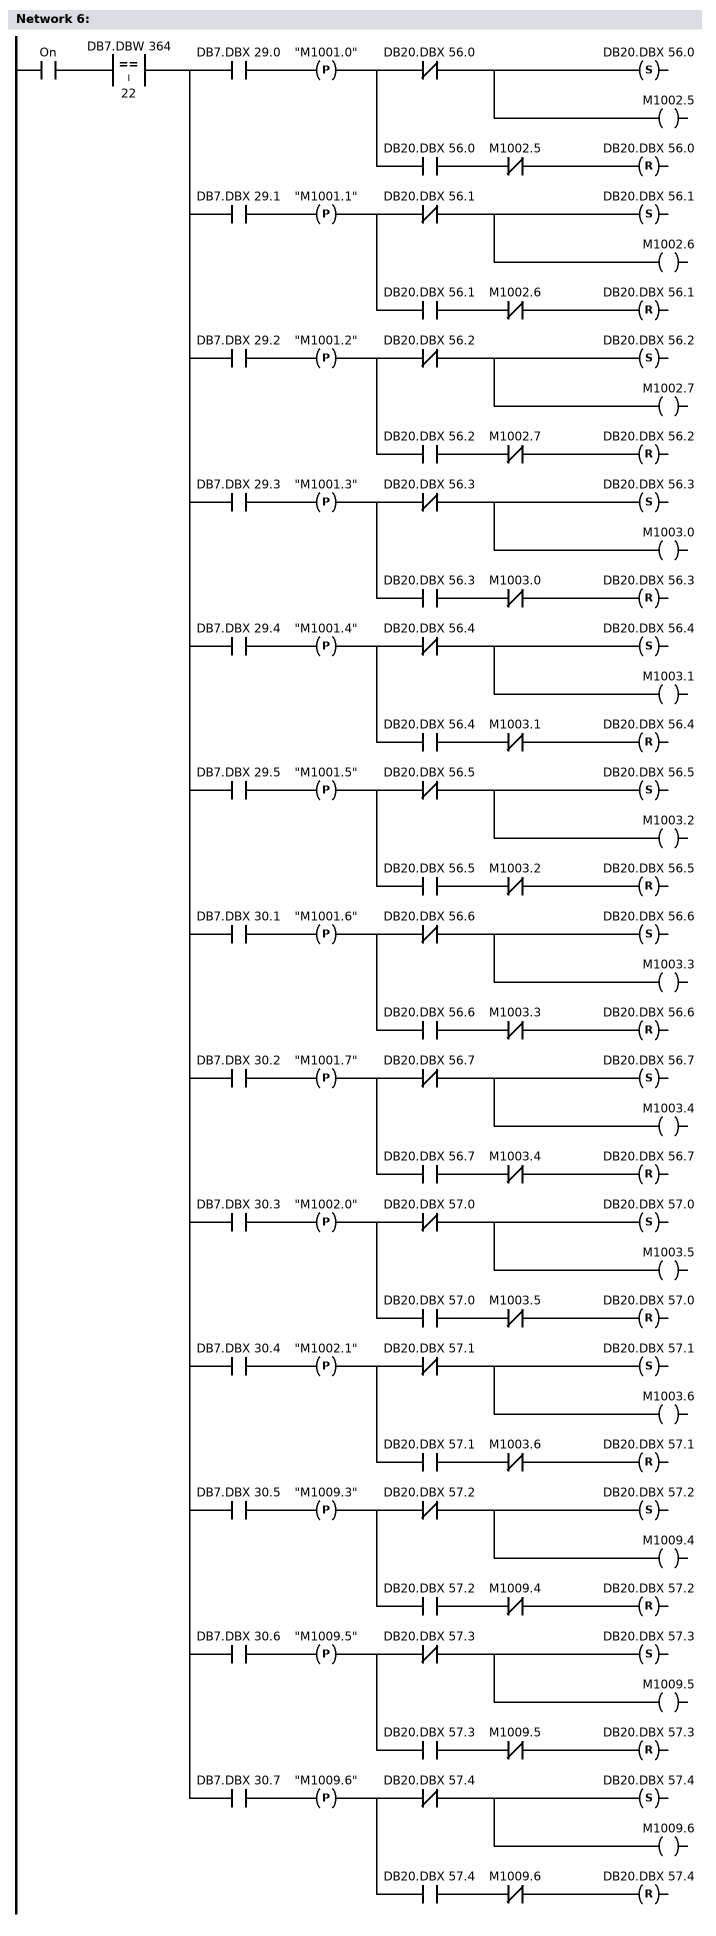
[picture p72: FC53 - REWORK networks 6-6]
NETWORK
TITLE =
      A     "On";
      A(;
      L     DB7.DBW 364;
      L     22;
      ==I;
      );
      =     L 0.0;
      A     L 0.0;
      A     DB7.DBX 29.0;
      FP    "M1001.0";
      =     L 0.1;
      A     L 0.1;
      AN    DB20.DBX 56.0;
      S     DB20.DBX 56.0;
      =     "M1002.5";
      A     L 0.1;
      A     DB20.DBX 56.0;
      AN    "M1002.5";
      R     DB20.DBX 56.0;
      A     L 0.0;
      A     DB7.DBX 29.1;
      FP    "M1001.1";
      =     L 0.1;
      A     L 0.1;
      AN    DB20.DBX 56.1;
      S     DB20.DBX 56.1;
      =     "M1002.6";
      A     L 0.1;
      A     DB20.DBX 56.1;
      AN    "M1002.6";
      R     DB20.DBX 56.1;
      A     L 0.0;
      A     DB7.DBX 29.2;
      FP    "M1001.2";
      =     L 0.1;
      A     L 0.1;
      AN    DB20.DBX 56.2;
      S     DB20.DBX 56.2;
      =     "M1002.7";
      A     L 0.1;
      A     DB20.DBX 56.2;
      AN    "M1002.7";
      R     DB20.DBX 56.2;
      A     L 0.0;
      A     DB7.DBX 29.3;
      FP    "M1001.3";
      =     L 0.1;
      A     L 0.1;
      AN    DB20.DBX 56.3;
      S     DB20.DBX 56.3;
      =     "M1003.0";
      A     L 0.1;
      A     DB20.DBX 56.3;
      AN    "M1003.0";
      R     DB20.DBX 56.3;
      A     L 0.0;
      A     DB7.DBX 29.4;
      FP    "M1001.4";
      =     L 0.1;
      A     L 0.1;
      AN    DB20.DBX 56.4;
      S     DB20.DBX 56.4;
      =     "M1003.1";
      A     L 0.1;
      A     DB20.DBX 56.4;
      AN    "M1003.1";
      R     DB20.DBX 56.4;
      A     L 0.0;
      A     DB7.DBX 29.5;
      FP    "M1001.5";
      =     L 0.1;
      A     L 0.1;
      AN    DB20.DBX 56.5;
      S     DB20.DBX 56.5;
      =     "M1003.2";
      A     L 0.1;
      A     DB20.DBX 56.5;
      AN    "M1003.2";
      R     DB20.DBX 56.5;
      A     L 0.0;
      A     DB7.DBX 30.1;
      FP    "M1001.6";
      =     L 0.1;
      A     L 0.1;
      AN    DB20.DBX 56.6;
      S     DB20.DBX 56.6;
      =     "M1003.3";
      A     L 0.1;
      A     DB20.DBX 56.6;
      AN    "M1003.3";
      R     DB20.DBX 56.6;
      A     L 0.0;
      A     DB7.DBX 30.2;
      FP    "M1001.7";
      =     L 0.1;
      A     L 0.1;
      AN    DB20.DBX 56.7;
      S     DB20.DBX 56.7;
      =     "M1003.4";
      A     L 0.1;
      A     DB20.DBX 56.7;
      AN    "M1003.4";
      R     DB20.DBX 56.7;
      A     L 0.0;
      A     DB7.DBX 30.3;
      FP    "M1002.0";
      =     L 0.1;
      A     L 0.1;
      AN    DB20.DBX 57.0;
      S     DB20.DBX 57.0;
      =     "M1003.5";
      A     L 0.1;
      A     DB20.DBX 57.0;
      AN    "M1003.5";
      R     DB20.DBX 57.0;
      A     L 0.0;
      A     DB7.DBX 30.4;
      FP    "M1002.1";
      =     L 0.1;
      A     L 0.1;
      AN    DB20.DBX 57.1;
      S     DB20.DBX 57.1;
      =     "M1003.6";
      A     L 0.1;
      A     DB20.DBX 57.1;
      AN    "M1003.6";
      R     DB20.DBX 57.1;
      A     L 0.0;
      A     DB7.DBX 30.5;
      FP    "M1009.3";
      =     L 0.1;
      A     L 0.1;
      AN    DB20.DBX 57.2;
      S     DB20.DBX 57.2;
      =     "M1009.4";
      A     L 0.1;
      A     DB20.DBX 57.2;
      AN    "M1009.4";
      R     DB20.DBX 57.2;
      A     L 0.0;
      A     DB7.DBX 30.6;
      FP    "M1009.5";
      =     L 0.1;
      A     L 0.1;
      AN    DB20.DBX 57.3;
      S     DB20.DBX 57.3;
      =     "M1009.5";
      A     L 0.1;
      A     DB20.DBX 57.3;
      AN    "M1009.5";
      R     DB20.DBX 57.3;
      A     L 0.0;
      A     DB7.DBX 30.7;
      FP    "M1009.6";
      =     L 0.1;
      A     L 0.1;
      AN    DB20.DBX 57.4;
      S     DB20.DBX 57.4;
      =     "M1009.6";
      A     L 0.1;
      A     DB20.DBX 57.4;
      AN    "M1009.6";
      R     DB20.DBX 57.4;
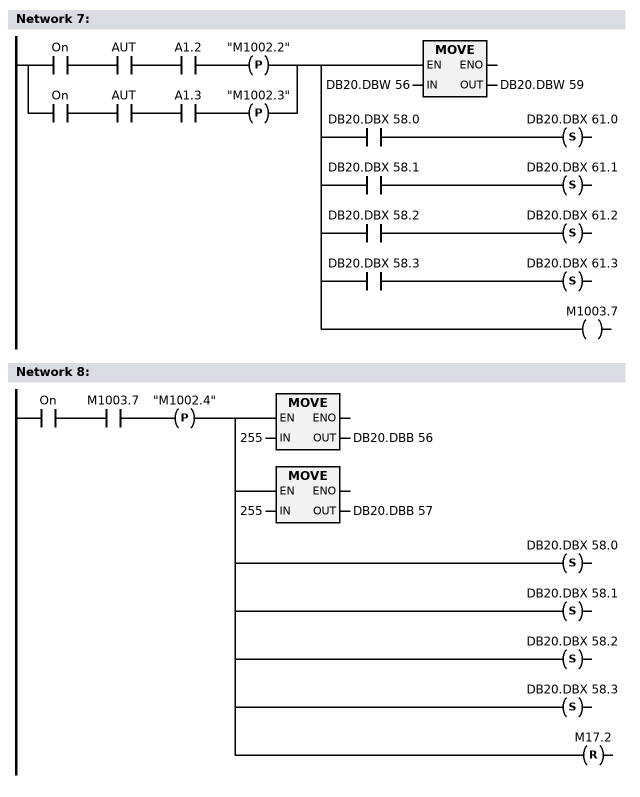
NETWORK
TITLE =
      A     "On";
      A     "AUT";
      A     "A1.2";
      FP    "M1002.2";
      O(;
      A     "On";
      A     "AUT";
      A     "A1.3";
      FP    "M1002.3";
      );
      =     L 0.0;
      A     L 0.0;
      JNB   M009;
      L     DB20.DBW 56;
      T     DB20.DBW 59;
M009: NOP   0;
      A     L 0.0;
      A     DB20.DBX 58.0;
      S     DB20.DBX 61.0;
      A     L 0.0;
      A     DB20.DBX 58.1;
      S     DB20.DBX 61.1;
      A     L 0.0;
      A     DB20.DBX 58.2;
      S     DB20.DBX 61.2;
      A     L 0.0;
      A     DB20.DBX 58.3;
      S     DB20.DBX 61.3;
      A     L 0.0;
      BLD   102;
      =     "M1003.7";
NETWORK
TITLE =
      A     "On";
      A     "M1003.7";
      FP    "M1002.4";
      =     L 0.0;
      A     L 0.0;
      JNB   M010;
      L     255;
      T     DB20.DBB 56;
M010: NOP   0;
      A     L 0.0;
      JNB   M011;
      L     255;
      T     DB20.DBB 57;
M011: NOP   0;
      A     L 0.0;
      BLD   102;
      S     DB20.DBX 58.0;
      A     L 0.0;
      BLD   102;
      S     DB20.DBX 58.1;
      A     L 0.0;
      BLD   102;
      S     DB20.DBX 58.2;
      A     L 0.0;
      BLD   102;
      S     DB20.DBX 58.3;
      A     L 0.0;
      BLD   102;
      R     "M17.2";
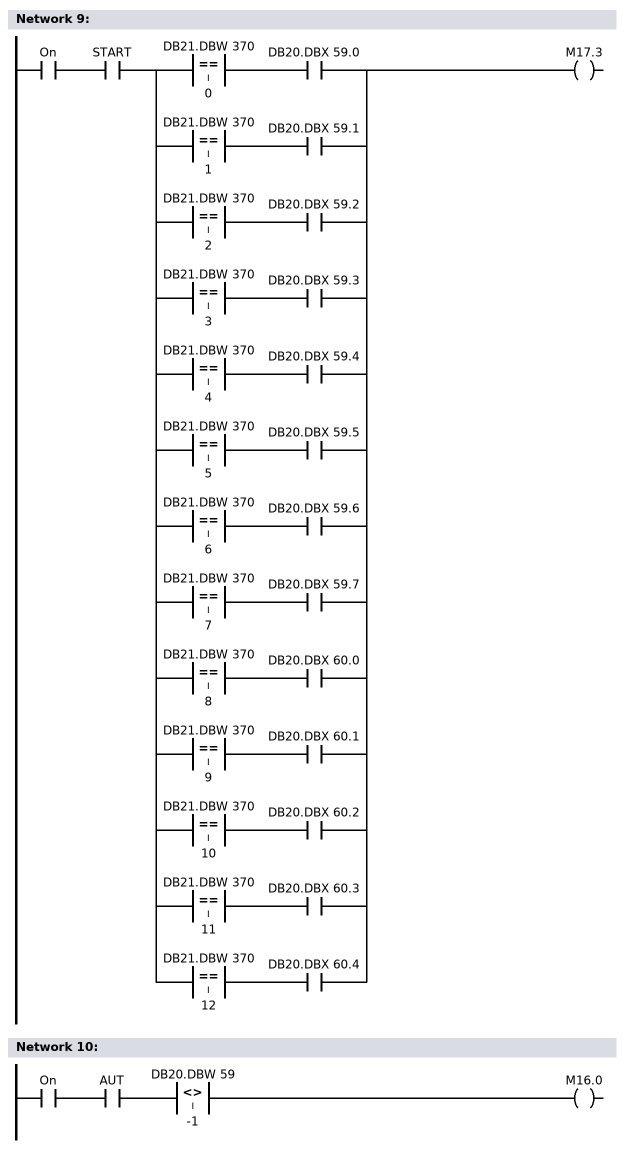
NETWORK
TITLE =
      A     "On";
      A     "START";
      A(;
      A(;
      L     DB21.DBW 370;
      L     0;
      ==I;
      );
      A     DB20.DBX 59.0;
      O;
      A(;
      L     DB21.DBW 370;
      L     1;
      ==I;
      );
      A     DB20.DBX 59.1;
      O;
      A(;
      L     DB21.DBW 370;
      L     2;
      ==I;
      );
      A     DB20.DBX 59.2;
      O;
      A(;
      L     DB21.DBW 370;
      L     3;
      ==I;
      );
      A     DB20.DBX 59.3;
      O;
      A(;
      L     DB21.DBW 370;
      L     4;
      ==I;
      );
      A     DB20.DBX 59.4;
      O;
      A(;
      L     DB21.DBW 370;
      L     5;
      ==I;
      );
      A     DB20.DBX 59.5;
      O;
      A(;
      L     DB21.DBW 370;
      L     6;
      ==I;
      );
      A     DB20.DBX 59.6;
      O;
      A(;
      L     DB21.DBW 370;
      L     7;
      ==I;
      );
      A     DB20.DBX 59.7;
      O;
      A(;
      L     DB21.DBW 370;
      L     8;
      ==I;
      );
      A     DB20.DBX 60.0;
      O;
      A(;
      L     DB21.DBW 370;
      L     9;
      ==I;
      );
      A     DB20.DBX 60.1;
      O;
      A(;
      L     DB21.DBW 370;
      L     10;
      ==I;
      );
      A     DB20.DBX 60.2;
      O;
      A(;
      L     DB21.DBW 370;
      L     11;
      ==I;
      );
      A     DB20.DBX 60.3;
      O;
      A(;
      L     DB21.DBW 370;
      L     12;
      ==I;
      );
      A     DB20.DBX 60.4;
      );
      =     "M17.3";
NETWORK
TITLE =
      A     "On";
      A     "AUT";
      A(;
      L     DB20.DBW 59;
      L     -1;
      <>I;
      );
      =     "M16.0";
END_FUNCTION

FUNCTION FC 54 : VOID
VERSION : 0.1
BEGIN
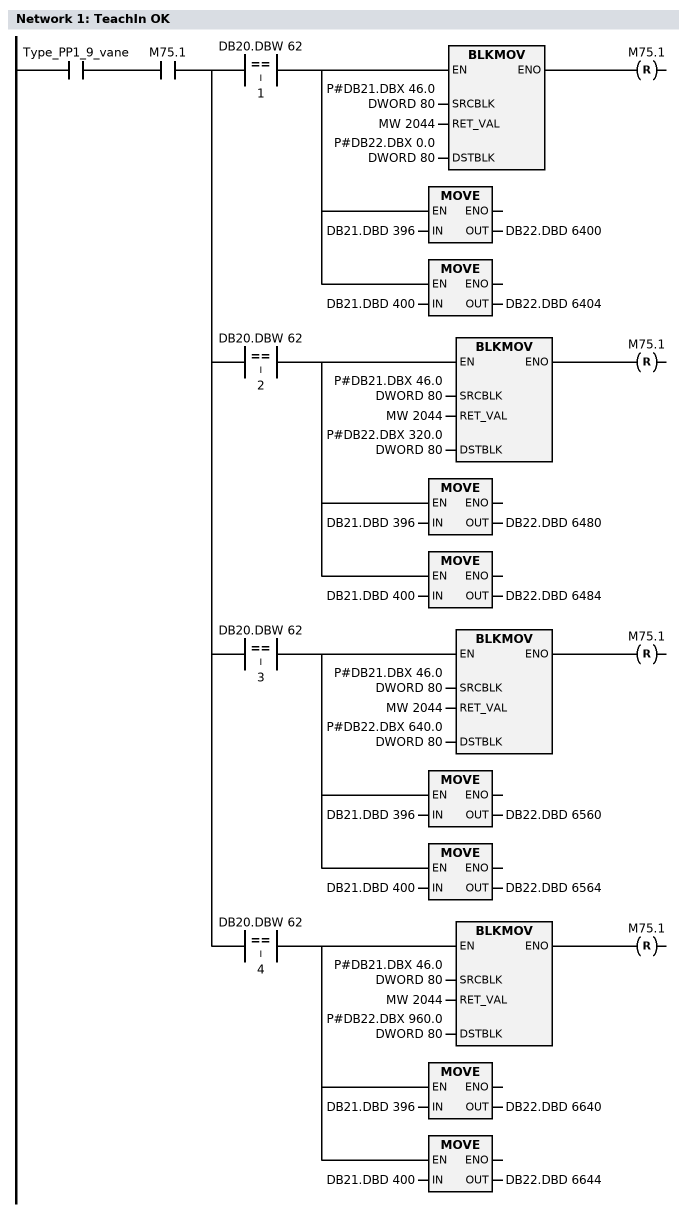
NETWORK
TITLE = TeachIn OK
      A     "Type_PP1_9_vane";
      A     "M75.1";
      =     L 0.0;
      A     L 0.0;
      A(;
      L     DB20.DBW 62;
      L     1;
      ==I;
      );
      =     L 0.1;
      A     L 0.1;
      JNB   _001;
      CALL  "BLKMOV" (
           SRCBLK                   := P#DB21.DBX 46.0 DWORD 80,
           RET_VAL                  := MW 2044,
           DSTBLK                   := P#DB22.DBX 0.0 DWORD 80);
_001: A     BR;
      R     "M75.1";
      A     L 0.1;
      JNB   _002;
      L     DB21.DBD 396;
      T     DB22.DBD 6400;
_002: NOP   0;
      A     L 0.1;
      JNB   _003;
      L     DB21.DBD 400;
      T     DB22.DBD 6404;
_003: NOP   0;
      A     L 0.0;
      A(;
      L     DB20.DBW 62;
      L     2;
      ==I;
      );
      =     L 0.1;
      A     L 0.1;
      JNB   _004;
      CALL  "BLKMOV" (
           SRCBLK                   := P#DB21.DBX 46.0 DWORD 80,
           RET_VAL                  := MW 2044,
           DSTBLK                   := P#DB22.DBX 320.0 DWORD 80);
_004: A     BR;
      R     "M75.1";
      A     L 0.1;
      JNB   _005;
      L     DB21.DBD 396;
      T     DB22.DBD 6480;
_005: NOP   0;
      A     L 0.1;
      JNB   _006;
      L     DB21.DBD 400;
      T     DB22.DBD 6484;
_006: NOP   0;
      A     L 0.0;
      A(;
      L     DB20.DBW 62;
      L     3;
      ==I;
      );
      =     L 0.1;
      A     L 0.1;
      JNB   _007;
      CALL  "BLKMOV" (
           SRCBLK                   := P#DB21.DBX 46.0 DWORD 80,
           RET_VAL                  := MW 2044,
           DSTBLK                   := P#DB22.DBX 640.0 DWORD 80);
_007: A     BR;
      R     "M75.1";
      A     L 0.1;
      JNB   _008;
      L     DB21.DBD 396;
      T     DB22.DBD 6560;
_008: NOP   0;
      A     L 0.1;
      JNB   _009;
      L     DB21.DBD 400;
      T     DB22.DBD 6564;
_009: NOP   0;
      A     L 0.0;
      A(;
      L     DB20.DBW 62;
      L     4;
      ==I;
      );
      =     L 0.1;
      A     L 0.1;
      JNB   _00a;
      CALL  "BLKMOV" (
           SRCBLK                   := P#DB21.DBX 46.0 DWORD 80,
           RET_VAL                  := MW 2044,
           DSTBLK                   := P#DB22.DBX 960.0 DWORD 80);
_00a: A     BR;
      R     "M75.1";
      A     L 0.1;
      JNB   _00b;
      L     DB21.DBD 396;
      T     DB22.DBD 6640;
_00b: NOP   0;
      A     L 0.1;
      JNB   _00c;
      L     DB21.DBD 400;
      T     DB22.DBD 6644;
_00c: NOP   0;
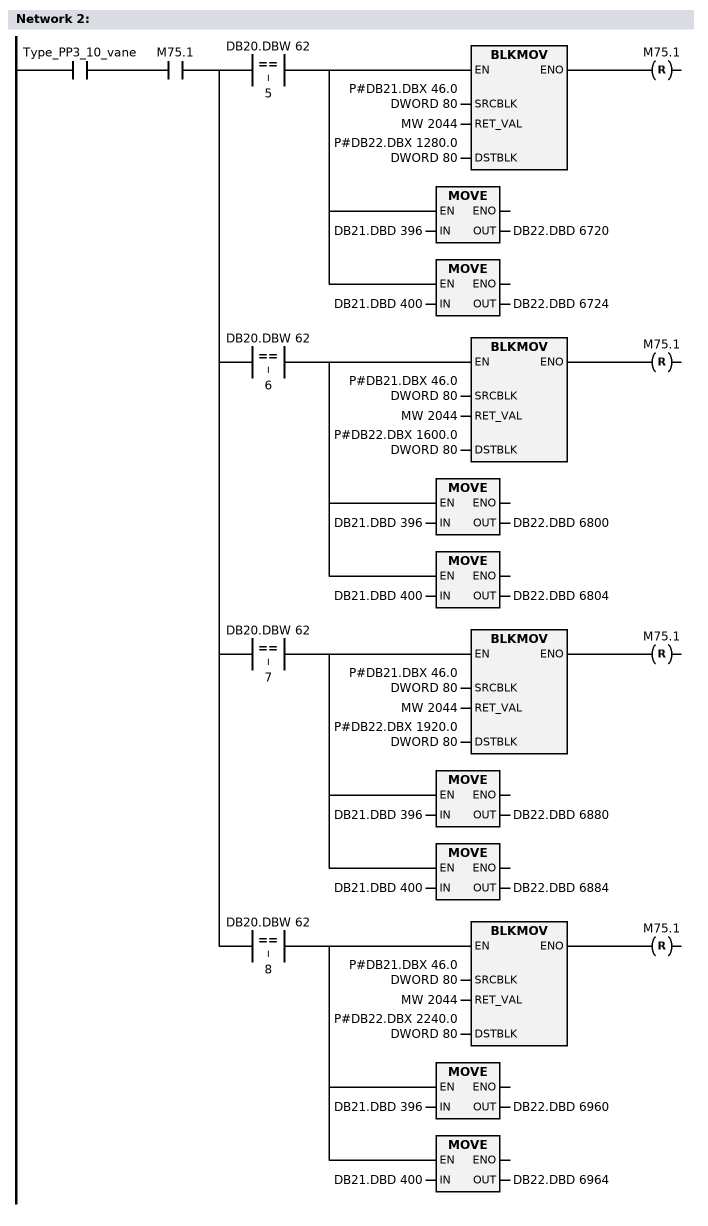
NETWORK
TITLE =
      A     "Type_PP3_10_vane";
      A     "M75.1";
      =     L 0.0;
      A     L 0.0;
      A(;
      L     DB20.DBW 62;
      L     5;
      ==I;
      );
      =     L 0.1;
      A     L 0.1;
      JNB   _00d;
      CALL  "BLKMOV" (
           SRCBLK                   := P#DB21.DBX 46.0 DWORD 80,
           RET_VAL                  := MW 2044,
           DSTBLK                   := P#DB22.DBX 1280.0 DWORD 80);
_00d: A     BR;
      R     "M75.1";
      A     L 0.1;
      JNB   _00e;
      L     DB21.DBD 396;
      T     DB22.DBD 6720;
_00e: NOP   0;
      A     L 0.1;
      JNB   _00f;
      L     DB21.DBD 400;
      T     DB22.DBD 6724;
_00f: NOP   0;
      A     L 0.0;
      A(;
      L     DB20.DBW 62;
      L     6;
      ==I;
      );
      =     L 0.1;
      A     L 0.1;
      JNB   _010;
      CALL  "BLKMOV" (
           SRCBLK                   := P#DB21.DBX 46.0 DWORD 80,
           RET_VAL                  := MW 2044,
           DSTBLK                   := P#DB22.DBX 1600.0 DWORD 80);
_010: A     BR;
      R     "M75.1";
      A     L 0.1;
      JNB   _011;
      L     DB21.DBD 396;
      T     DB22.DBD 6800;
_011: NOP   0;
      A     L 0.1;
      JNB   _012;
      L     DB21.DBD 400;
      T     DB22.DBD 6804;
_012: NOP   0;
      A     L 0.0;
      A(;
      L     DB20.DBW 62;
      L     7;
      ==I;
      );
      =     L 0.1;
      A     L 0.1;
      JNB   _013;
      CALL  "BLKMOV" (
           SRCBLK                   := P#DB21.DBX 46.0 DWORD 80,
           RET_VAL                  := MW 2044,
           DSTBLK                   := P#DB22.DBX 1920.0 DWORD 80);
_013: A     BR;
      R     "M75.1";
      A     L 0.1;
      JNB   _014;
      L     DB21.DBD 396;
      T     DB22.DBD 6880;
_014: NOP   0;
      A     L 0.1;
      JNB   _015;
      L     DB21.DBD 400;
      T     DB22.DBD 6884;
_015: NOP   0;
      A     L 0.0;
      A(;
      L     DB20.DBW 62;
      L     8;
      ==I;
      );
      =     L 0.1;
      A     L 0.1;
      JNB   _016;
      CALL  "BLKMOV" (
           SRCBLK                   := P#DB21.DBX 46.0 DWORD 80,
           RET_VAL                  := MW 2044,
           DSTBLK                   := P#DB22.DBX 2240.0 DWORD 80);
_016: A     BR;
      R     "M75.1";
      A     L 0.1;
      JNB   _017;
      L     DB21.DBD 396;
      T     DB22.DBD 6960;
_017: NOP   0;
      A     L 0.1;
      JNB   _018;
      L     DB21.DBD 400;
      T     DB22.DBD 6964;
_018: NOP   0;
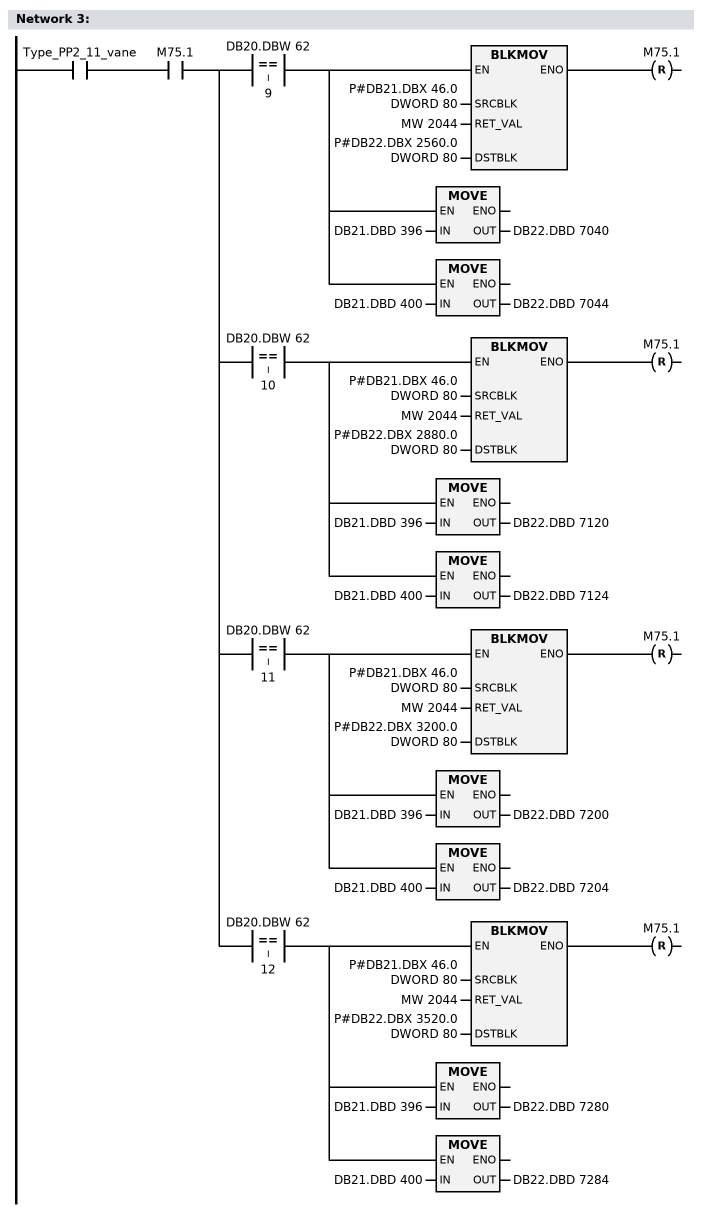
NETWORK
TITLE =
      A     "Type_PP2_11_vane";
      A     "M75.1";
      =     L 0.0;
      A     L 0.0;
      A(;
      L     DB20.DBW 62;
      L     9;
      ==I;
      );
      =     L 0.1;
      A     L 0.1;
      JNB   _019;
      CALL  "BLKMOV" (
           SRCBLK                   := P#DB21.DBX 46.0 DWORD 80,
           RET_VAL                  := MW 2044,
           DSTBLK                   := P#DB22.DBX 2560.0 DWORD 80);
_019: A     BR;
      R     "M75.1";
      A     L 0.1;
      JNB   _01a;
      L     DB21.DBD 396;
      T     DB22.DBD 7040;
_01a: NOP   0;
      A     L 0.1;
      JNB   _01b;
      L     DB21.DBD 400;
      T     DB22.DBD 7044;
_01b: NOP   0;
      A     L 0.0;
      A(;
      L     DB20.DBW 62;
      L     10;
      ==I;
      );
      =     L 0.1;
      A     L 0.1;
      JNB   _01c;
      CALL  "BLKMOV" (
           SRCBLK                   := P#DB21.DBX 46.0 DWORD 80,
           RET_VAL                  := MW 2044,
           DSTBLK                   := P#DB22.DBX 2880.0 DWORD 80);
_01c: A     BR;
      R     "M75.1";
      A     L 0.1;
      JNB   _01d;
      L     DB21.DBD 396;
      T     DB22.DBD 7120;
_01d: NOP   0;
      A     L 0.1;
      JNB   _01e;
      L     DB21.DBD 400;
      T     DB22.DBD 7124;
_01e: NOP   0;
      A     L 0.0;
      A(;
      L     DB20.DBW 62;
      L     11;
      ==I;
      );
      =     L 0.1;
      A     L 0.1;
      JNB   _01f;
      CALL  "BLKMOV" (
           SRCBLK                   := P#DB21.DBX 46.0 DWORD 80,
           RET_VAL                  := MW 2044,
           DSTBLK                   := P#DB22.DBX 3200.0 DWORD 80);
_01f: A     BR;
      R     "M75.1";
      A     L 0.1;
      JNB   _020;
      L     DB21.DBD 396;
      T     DB22.DBD 7200;
_020: NOP   0;
      A     L 0.1;
      JNB   _021;
      L     DB21.DBD 400;
      T     DB22.DBD 7204;
_021: NOP   0;
      A     L 0.0;
      A(;
      L     DB20.DBW 62;
      L     12;
      ==I;
      );
      =     L 0.1;
      A     L 0.1;
      JNB   _022;
      CALL  "BLKMOV" (
           SRCBLK                   := P#DB21.DBX 46.0 DWORD 80,
           RET_VAL                  := MW 2044,
           DSTBLK                   := P#DB22.DBX 3520.0 DWORD 80);
_022: A     BR;
      R     "M75.1";
      A     L 0.1;
      JNB   _023;
      L     DB21.DBD 396;
      T     DB22.DBD 7280;
_023: NOP   0;
      A     L 0.1;
      JNB   _024;
      L     DB21.DBD 400;
      T     DB22.DBD 7284;
_024: NOP   0;
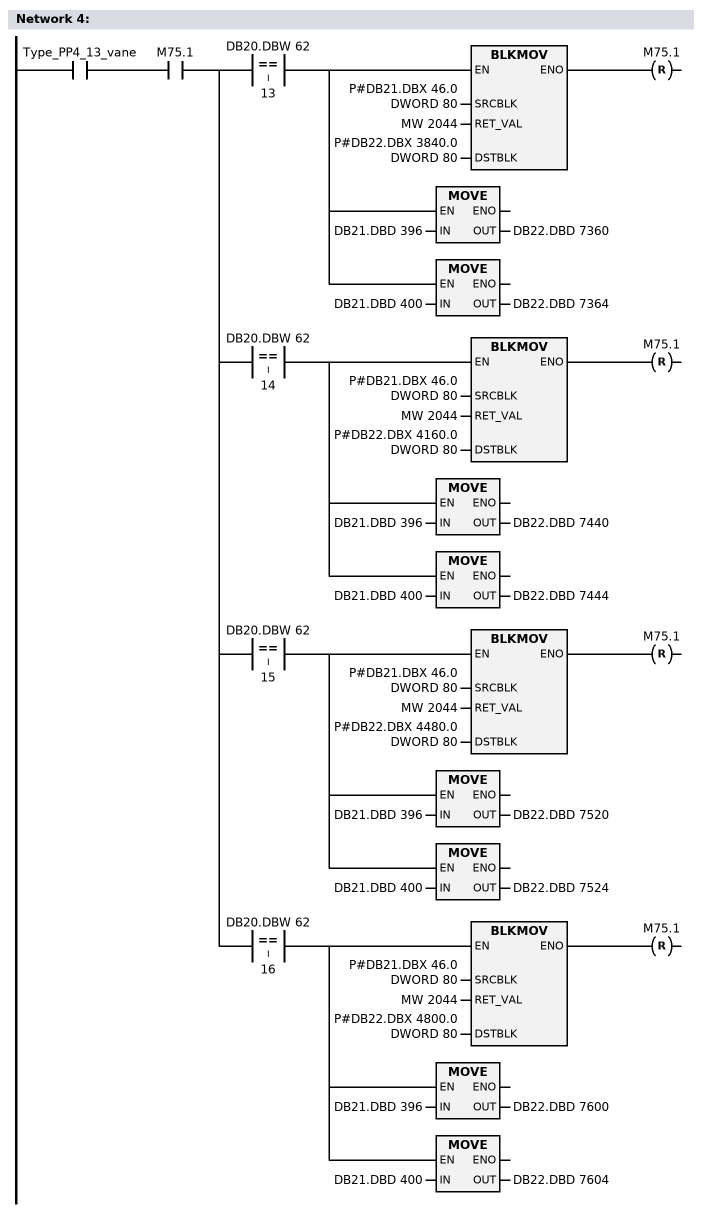
NETWORK
TITLE =
      A     "Type_PP4_13_vane";
      A     "M75.1";
      =     L 0.0;
      A     L 0.0;
      A(;
      L     DB20.DBW 62;
      L     13;
      ==I;
      );
      =     L 0.1;
      A     L 0.1;
      JNB   _025;
      CALL  "BLKMOV" (
           SRCBLK                   := P#DB21.DBX 46.0 DWORD 80,
           RET_VAL                  := MW 2044,
           DSTBLK                   := P#DB22.DBX 3840.0 DWORD 80);
_025: A     BR;
      R     "M75.1";
      A     L 0.1;
      JNB   _026;
      L     DB21.DBD 396;
      T     DB22.DBD 7360;
_026: NOP   0;
      A     L 0.1;
      JNB   _027;
      L     DB21.DBD 400;
      T     DB22.DBD 7364;
_027: NOP   0;
      A     L 0.0;
      A(;
      L     DB20.DBW 62;
      L     14;
      ==I;
      );
      =     L 0.1;
      A     L 0.1;
      JNB   _028;
      CALL  "BLKMOV" (
           SRCBLK                   := P#DB21.DBX 46.0 DWORD 80,
           RET_VAL                  := MW 2044,
           DSTBLK                   := P#DB22.DBX 4160.0 DWORD 80);
_028: A     BR;
      R     "M75.1";
      A     L 0.1;
      JNB   _029;
      L     DB21.DBD 396;
      T     DB22.DBD 7440;
_029: NOP   0;
      A     L 0.1;
      JNB   _02a;
      L     DB21.DBD 400;
      T     DB22.DBD 7444;
_02a: NOP   0;
      A     L 0.0;
      A(;
      L     DB20.DBW 62;
      L     15;
      ==I;
      );
      =     L 0.1;
      A     L 0.1;
      JNB   _02b;
      CALL  "BLKMOV" (
           SRCBLK                   := P#DB21.DBX 46.0 DWORD 80,
           RET_VAL                  := MW 2044,
           DSTBLK                   := P#DB22.DBX 4480.0 DWORD 80);
_02b: A     BR;
      R     "M75.1";
      A     L 0.1;
      JNB   _02c;
      L     DB21.DBD 396;
      T     DB22.DBD 7520;
_02c: NOP   0;
      A     L 0.1;
      JNB   _02d;
      L     DB21.DBD 400;
      T     DB22.DBD 7524;
_02d: NOP   0;
      A     L 0.0;
      A(;
      L     DB20.DBW 62;
      L     16;
      ==I;
      );
      =     L 0.1;
      A     L 0.1;
      JNB   _02e;
      CALL  "BLKMOV" (
           SRCBLK                   := P#DB21.DBX 46.0 DWORD 80,
           RET_VAL                  := MW 2044,
           DSTBLK                   := P#DB22.DBX 4800.0 DWORD 80);
_02e: A     BR;
      R     "M75.1";
      A     L 0.1;
      JNB   _02f;
      L     DB21.DBD 396;
      T     DB22.DBD 7600;
_02f: NOP   0;
      A     L 0.1;
      JNB   _030;
      L     DB21.DBD 400;
      T     DB22.DBD 7604;
_030: NOP   0;
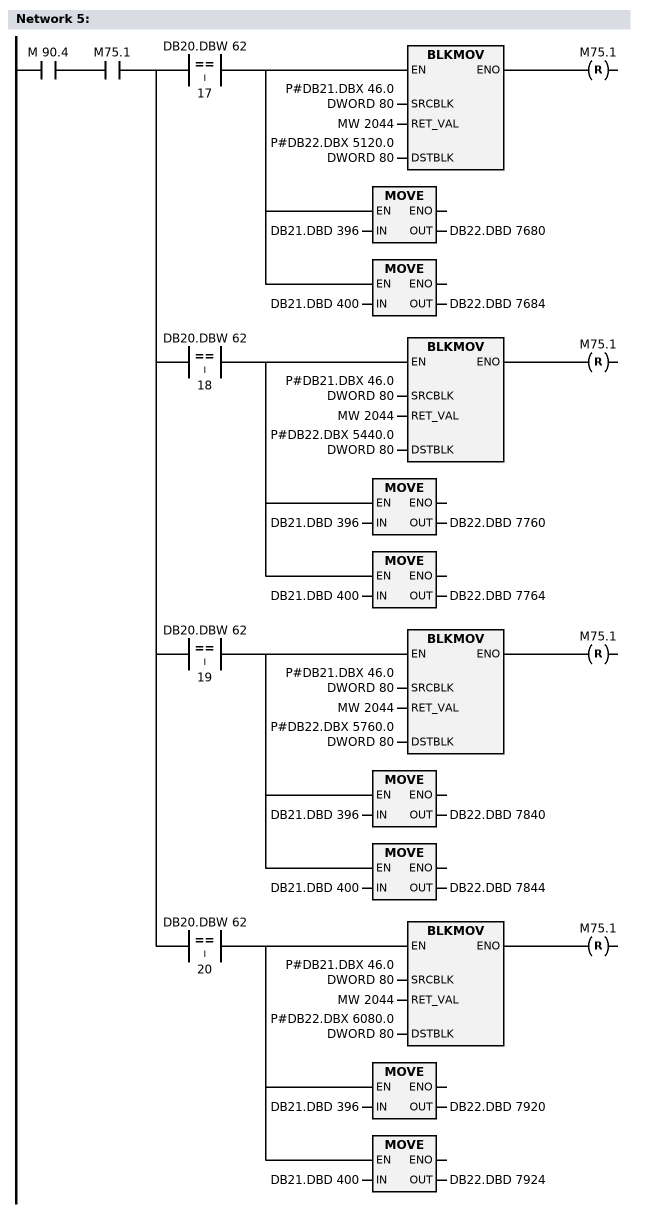
NETWORK
TITLE =
      A     M 90.4;
      A     "M75.1";
      =     L 0.0;
      A     L 0.0;
      A(;
      L     DB20.DBW 62;
      L     17;
      ==I;
      );
      =     L 0.1;
      A     L 0.1;
      JNB   _031;
      CALL  "BLKMOV" (
           SRCBLK                   := P#DB21.DBX 46.0 DWORD 80,
           RET_VAL                  := MW 2044,
           DSTBLK                   := P#DB22.DBX 5120.0 DWORD 80);
_031: A     BR;
      R     "M75.1";
      A     L 0.1;
      JNB   _032;
      L     DB21.DBD 396;
      T     DB22.DBD 7680;
_032: NOP   0;
      A     L 0.1;
      JNB   _033;
      L     DB21.DBD 400;
      T     DB22.DBD 7684;
_033: NOP   0;
      A     L 0.0;
      A(;
      L     DB20.DBW 62;
      L     18;
      ==I;
      );
      =     L 0.1;
      A     L 0.1;
      JNB   _034;
      CALL  "BLKMOV" (
           SRCBLK                   := P#DB21.DBX 46.0 DWORD 80,
           RET_VAL                  := MW 2044,
           DSTBLK                   := P#DB22.DBX 5440.0 DWORD 80);
_034: A     BR;
      R     "M75.1";
      A     L 0.1;
      JNB   _035;
      L     DB21.DBD 396;
      T     DB22.DBD 7760;
_035: NOP   0;
      A     L 0.1;
      JNB   _036;
      L     DB21.DBD 400;
      T     DB22.DBD 7764;
_036: NOP   0;
      A     L 0.0;
      A(;
      L     DB20.DBW 62;
      L     19;
      ==I;
      );
      =     L 0.1;
      A     L 0.1;
      JNB   _037;
      CALL  "BLKMOV" (
           SRCBLK                   := P#DB21.DBX 46.0 DWORD 80,
           RET_VAL                  := MW 2044,
           DSTBLK                   := P#DB22.DBX 5760.0 DWORD 80);
_037: A     BR;
      R     "M75.1";
      A     L 0.1;
      JNB   _038;
      L     DB21.DBD 396;
      T     DB22.DBD 7840;
_038: NOP   0;
      A     L 0.1;
      JNB   _039;
      L     DB21.DBD 400;
      T     DB22.DBD 7844;
_039: NOP   0;
      A     L 0.0;
      A(;
      L     DB20.DBW 62;
      L     20;
      ==I;
      );
      =     L 0.1;
      A     L 0.1;
      JNB   _03a;
      CALL  "BLKMOV" (
           SRCBLK                   := P#DB21.DBX 46.0 DWORD 80,
           RET_VAL                  := MW 2044,
           DSTBLK                   := P#DB22.DBX 6080.0 DWORD 80);
_03a: A     BR;
      R     "M75.1";
      A     L 0.1;
      JNB   _03b;
      L     DB21.DBD 396;
      T     DB22.DBD 7920;
_03b: NOP   0;
      A     L 0.1;
      JNB   _03c;
      L     DB21.DBD 400;
      T     DB22.DBD 7924;
_03c: NOP   0;
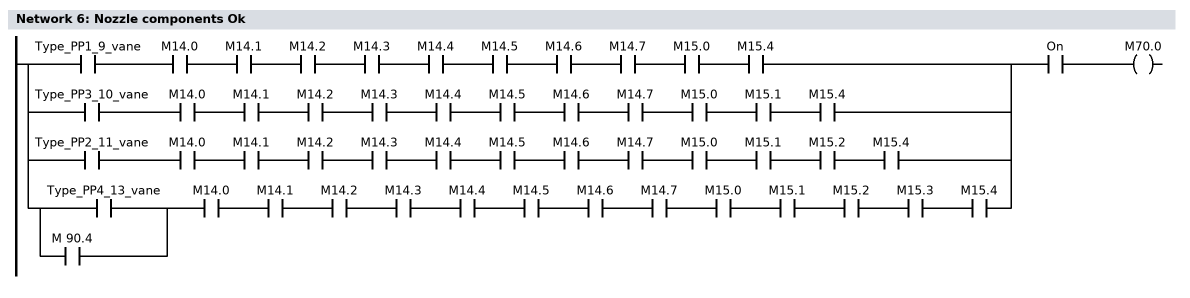
NETWORK
TITLE = Nozzle components Ok
      A(;
      A     "Type_PP1_9_vane";
      A     "M14.0";
      A     "M14.1";
      A     "M14.2";
      A     "M14.3";
      A     "M14.4";
      A     "M14.5";
      A     "M14.6";
      A     "M14.7";
      A     "M15.0";
      A     "M15.4";
      O;
      A     "Type_PP3_10_vane";
      A     "M14.0";
      A     "M14.1";
      A     "M14.2";
      A     "M14.3";
      A     "M14.4";
      A     "M14.5";
      A     "M14.6";
      A     "M14.7";
      A     "M15.0";
      A     "M15.1";
      A     "M15.4";
      O;
      A     "Type_PP2_11_vane";
      A     "M14.0";
      A     "M14.1";
      A     "M14.2";
      A     "M14.3";
      A     "M14.4";
      A     "M14.5";
      A     "M14.6";
      A     "M14.7";
      A     "M15.0";
      A     "M15.1";
      A     "M15.2";
      A     "M15.4";
      O;
      A(;
      O     "Type_PP4_13_vane";
      O     M 90.4;
      );
      A     "M14.0";
      A     "M14.1";
      A     "M14.2";
      A     "M14.3";
      A     "M14.4";
      A     "M14.5";
      A     "M14.6";
      A     "M14.7";
      A     "M15.0";
      A     "M15.1";
      A     "M15.2";
      A     "M15.3";
      A     "M15.4";
      );
      A     "On";
      =     "M70.0";
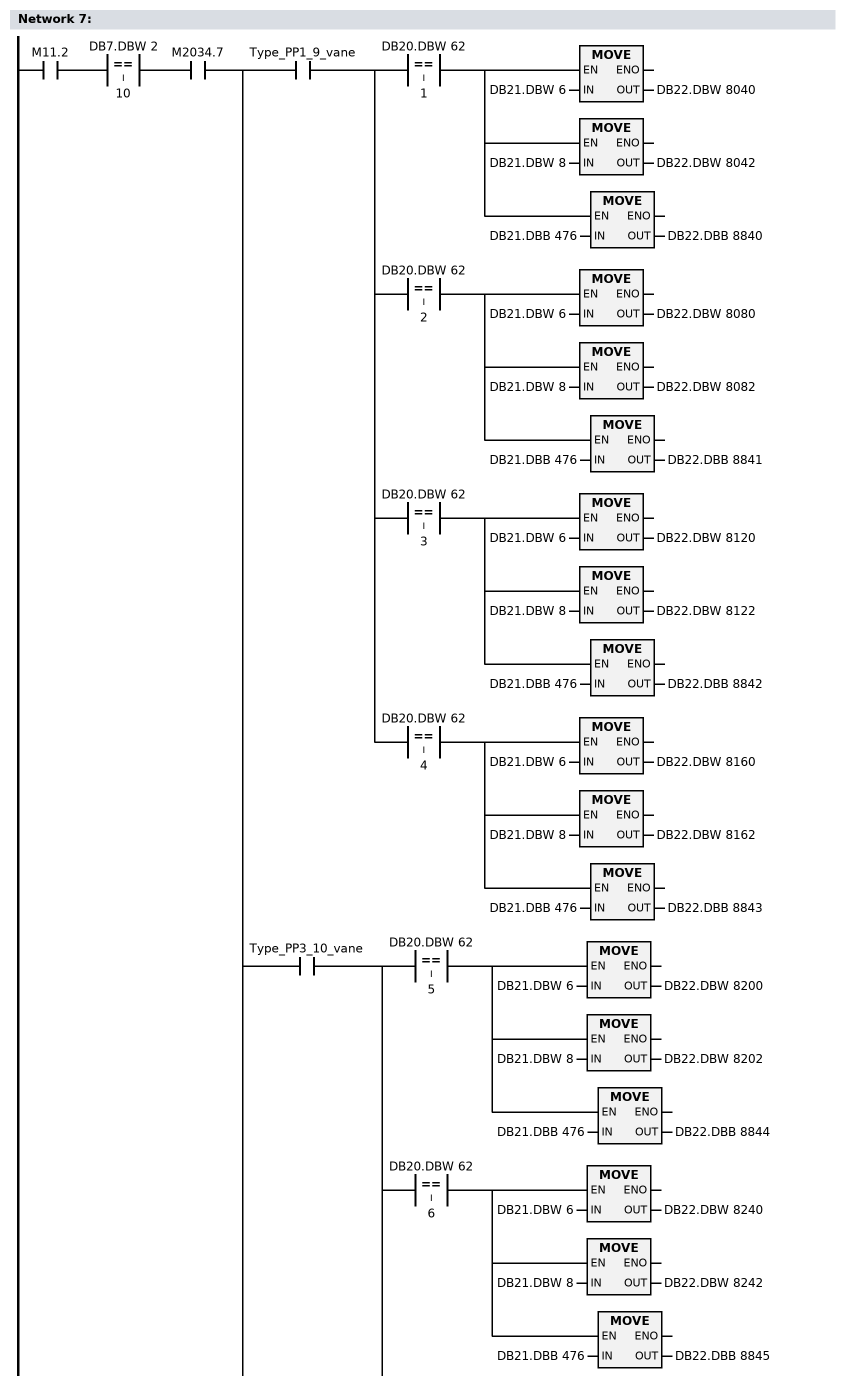
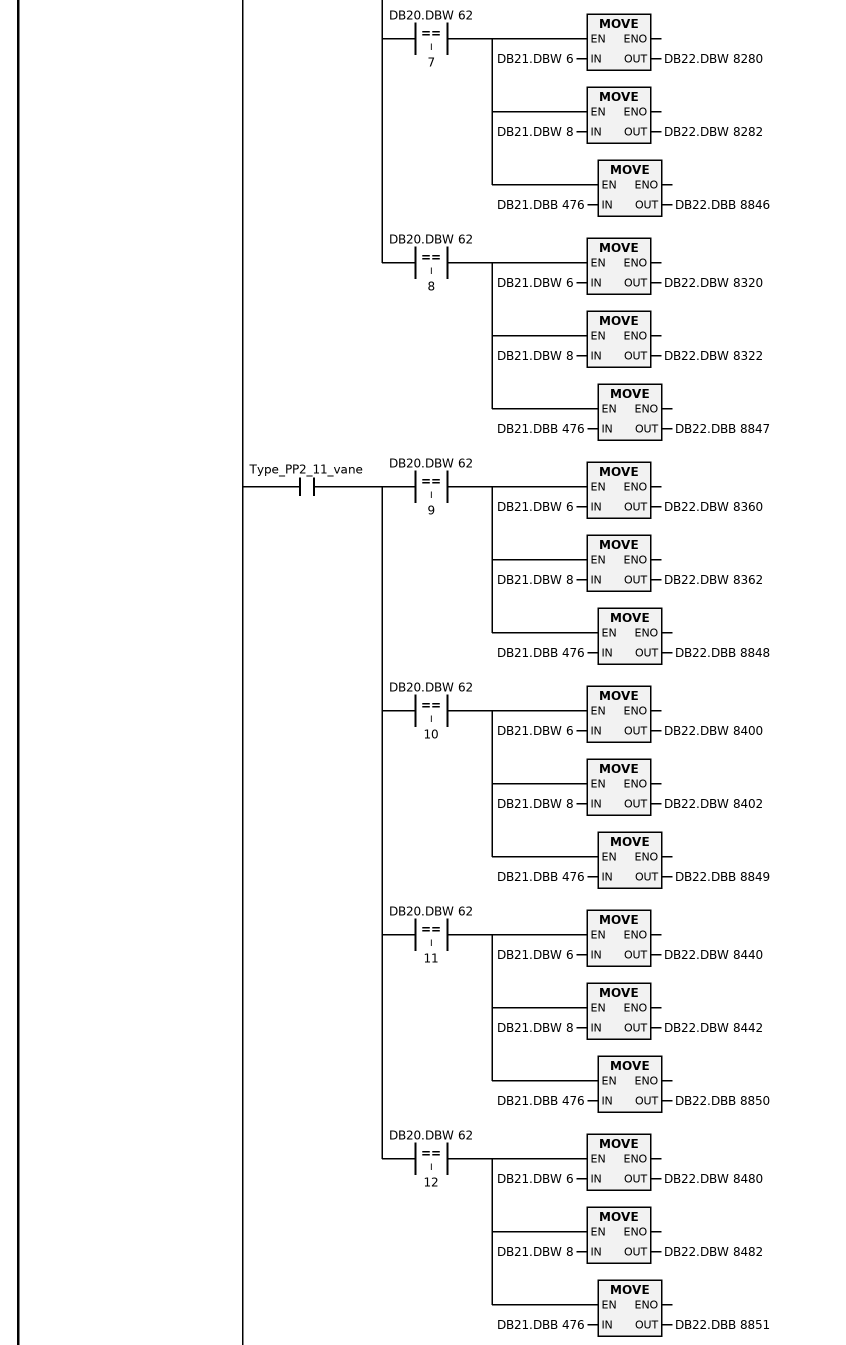
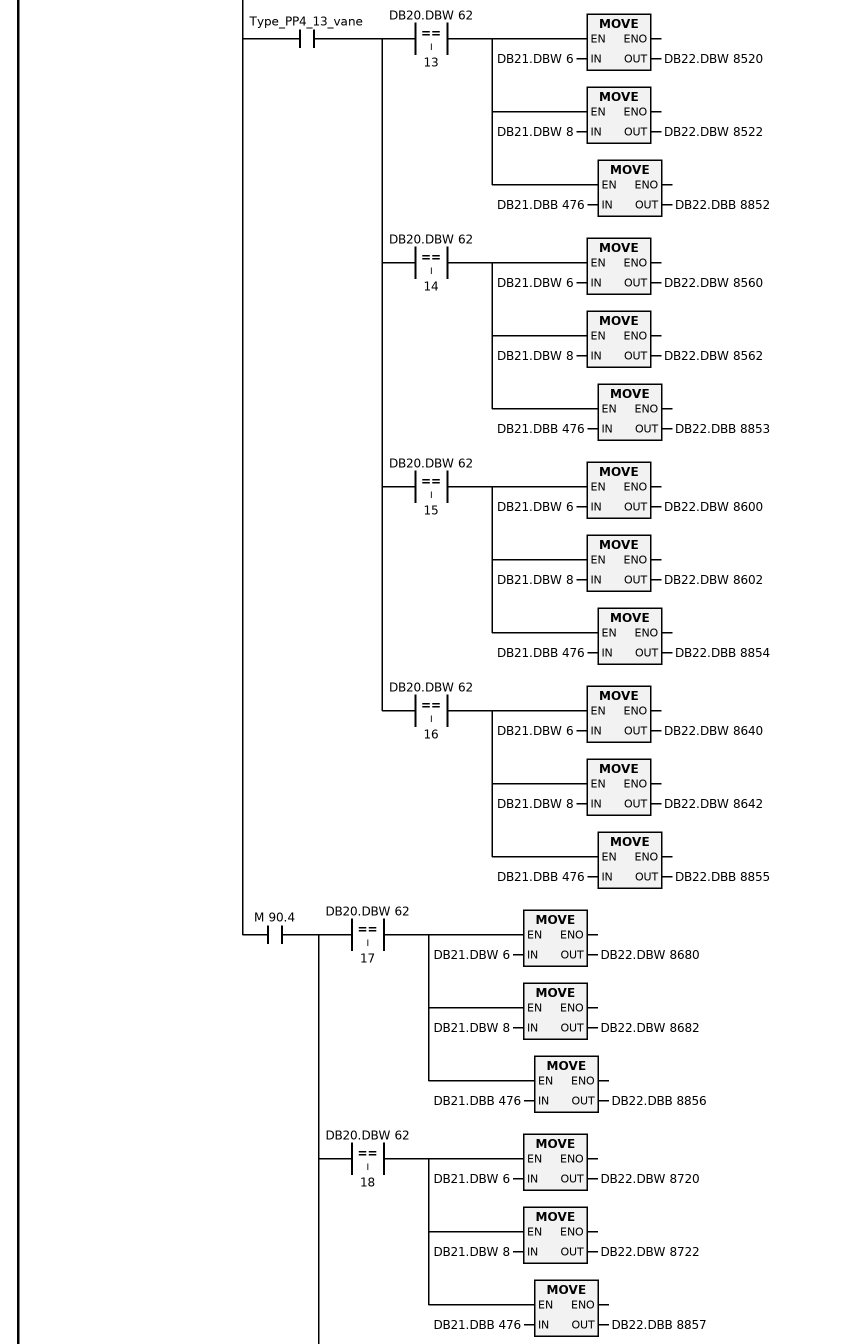
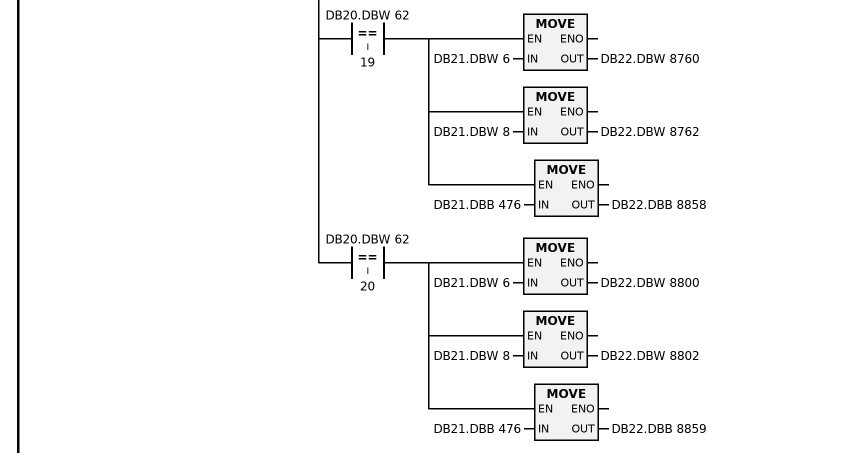
NETWORK
TITLE =
      A     "M11.2";
      A(;
      L     DB7.DBW 2;
      L     10;
      ==I;
      );
      A     "M2034.7";
      =     L 0.0;
      A     L 0.0;
      A     "Type_PP1_9_vane";
      =     L 0.1;
      A     L 0.1;
      A(;
      L     DB20.DBW 62;
      L     1;
      ==I;
      );
      =     L 0.2;
      A     L 0.2;
      JNB   _03d;
      L     DB21.DBW 6;
      T     DB22.DBW 8040;
_03d: NOP   0;
      A     L 0.2;
      JNB   _03e;
      L     DB21.DBW 8;
      T     DB22.DBW 8042;
_03e: NOP   0;
      A     L 0.2;
      JNB   _03f;
      L     DB21.DBB 476;
      T     DB22.DBB 8840;
_03f: NOP   0;
      A     L 0.1;
      A(;
      L     DB20.DBW 62;
      L     2;
      ==I;
      );
      =     L 0.2;
      A     L 0.2;
      JNB   _040;
      L     DB21.DBW 6;
      T     DB22.DBW 8080;
_040: NOP   0;
      A     L 0.2;
      JNB   _041;
      L     DB21.DBW 8;
      T     DB22.DBW 8082;
_041: NOP   0;
      A     L 0.2;
      JNB   _042;
      L     DB21.DBB 476;
      T     DB22.DBB 8841;
_042: NOP   0;
      A     L 0.1;
      A(;
      L     DB20.DBW 62;
      L     3;
      ==I;
      );
      =     L 0.2;
      A     L 0.2;
      JNB   _043;
      L     DB21.DBW 6;
      T     DB22.DBW 8120;
_043: NOP   0;
      A     L 0.2;
      JNB   _044;
      L     DB21.DBW 8;
      T     DB22.DBW 8122;
_044: NOP   0;
      A     L 0.2;
      JNB   _045;
      L     DB21.DBB 476;
      T     DB22.DBB 8842;
_045: NOP   0;
      A     L 0.1;
      A(;
      L     DB20.DBW 62;
      L     4;
      ==I;
      );
      =     L 0.2;
      A     L 0.2;
      JNB   _046;
      L     DB21.DBW 6;
      T     DB22.DBW 8160;
_046: NOP   0;
      A     L 0.2;
      JNB   _047;
      L     DB21.DBW 8;
      T     DB22.DBW 8162;
_047: NOP   0;
      A     L 0.2;
      JNB   _048;
      L     DB21.DBB 476;
      T     DB22.DBB 8843;
_048: NOP   0;
      A     L 0.0;
      A     "Type_PP3_10_vane";
      =     L 0.1;
      A     L 0.1;
      A(;
      L     DB20.DBW 62;
      L     5;
      ==I;
      );
      =     L 0.2;
      A     L 0.2;
      JNB   _049;
      L     DB21.DBW 6;
      T     DB22.DBW 8200;
_049: NOP   0;
      A     L 0.2;
      JNB   _04a;
      L     DB21.DBW 8;
      T     DB22.DBW 8202;
_04a: NOP   0;
      A     L 0.2;
      JNB   _04b;
      L     DB21.DBB 476;
      T     DB22.DBB 8844;
_04b: NOP   0;
      A     L 0.1;
      A(;
      L     DB20.DBW 62;
      L     6;
      ==I;
      );
      =     L 0.2;
      A     L 0.2;
      JNB   _04c;
      L     DB21.DBW 6;
      T     DB22.DBW 8240;
_04c: NOP   0;
      A     L 0.2;
      JNB   _04d;
      L     DB21.DBW 8;
      T     DB22.DBW 8242;
_04d: NOP   0;
      A     L 0.2;
      JNB   _04e;
      L     DB21.DBB 476;
      T     DB22.DBB 8845;
_04e: NOP   0;
      A     L 0.1;
      A(;
      L     DB20.DBW 62;
      L     7;
      ==I;
      );
      =     L 0.2;
      A     L 0.2;
      JNB   _04f;
      L     DB21.DBW 6;
      T     DB22.DBW 8280;
_04f: NOP   0;
      A     L 0.2;
      JNB   _050;
      L     DB21.DBW 8;
      T     DB22.DBW 8282;
_050: NOP   0;
      A     L 0.2;
      JNB   _051;
      L     DB21.DBB 476;
      T     DB22.DBB 8846;
_051: NOP   0;
      A     L 0.1;
      A(;
      L     DB20.DBW 62;
      L     8;
      ==I;
      );
      =     L 0.2;
      A     L 0.2;
      JNB   _052;
      L     DB21.DBW 6;
      T     DB22.DBW 8320;
_052: NOP   0;
      A     L 0.2;
      JNB   _053;
      L     DB21.DBW 8;
      T     DB22.DBW 8322;
_053: NOP   0;
      A     L 0.2;
      JNB   _054;
      L     DB21.DBB 476;
      T     DB22.DBB 8847;
_054: NOP   0;
      A     L 0.0;
      A     "Type_PP2_11_vane";
      =     L 0.1;
      A     L 0.1;
      A(;
      L     DB20.DBW 62;
      L     9;
      ==I;
      );
      =     L 0.2;
      A     L 0.2;
      JNB   _055;
      L     DB21.DBW 6;
      T     DB22.DBW 8360;
_055: NOP   0;
      A     L 0.2;
      JNB   _056;
      L     DB21.DBW 8;
      T     DB22.DBW 8362;
_056: NOP   0;
      A     L 0.2;
      JNB   _057;
      L     DB21.DBB 476;
      T     DB22.DBB 8848;
_057: NOP   0;
      A     L 0.1;
      A(;
      L     DB20.DBW 62;
      L     10;
      ==I;
      );
      =     L 0.2;
      A     L 0.2;
      JNB   _058;
      L     DB21.DBW 6;
      T     DB22.DBW 8400;
_058: NOP   0;
      A     L 0.2;
      JNB   _059;
      L     DB21.DBW 8;
      T     DB22.DBW 8402;
_059: NOP   0;
      A     L 0.2;
      JNB   _05a;
      L     DB21.DBB 476;
      T     DB22.DBB 8849;
_05a: NOP   0;
      A     L 0.1;
      A(;
      L     DB20.DBW 62;
      L     11;
      ==I;
      );
      =     L 0.2;
      A     L 0.2;
      JNB   _05b;
      L     DB21.DBW 6;
      T     DB22.DBW 8440;
_05b: NOP   0;
      A     L 0.2;
      JNB   _05c;
      L     DB21.DBW 8;
      T     DB22.DBW 8442;
_05c: NOP   0;
      A     L 0.2;
      JNB   _05d;
      L     DB21.DBB 476;
      T     DB22.DBB 8850;
_05d: NOP   0;
      A     L 0.1;
      A(;
      L     DB20.DBW 62;
      L     12;
      ==I;
      );
      =     L 0.2;
      A     L 0.2;
      JNB   _05e;
      L     DB21.DBW 6;
      T     DB22.DBW 8480;
_05e: NOP   0;
      A     L 0.2;
      JNB   _05f;
      L     DB21.DBW 8;
      T     DB22.DBW 8482;
_05f: NOP   0;
      A     L 0.2;
      JNB   _060;
      L     DB21.DBB 476;
      T     DB22.DBB 8851;
_060: NOP   0;
      A     L 0.0;
      A     "Type_PP4_13_vane";
      =     L 0.1;
      A     L 0.1;
      A(;
      L     DB20.DBW 62;
      L     13;
      ==I;
      );
      =     L 0.2;
      A     L 0.2;
      JNB   _061;
      L     DB21.DBW 6;
      T     DB22.DBW 8520;
_061: NOP   0;
      A     L 0.2;
      JNB   _062;
      L     DB21.DBW 8;
      T     DB22.DBW 8522;
_062: NOP   0;
      A     L 0.2;
      JNB   _063;
      L     DB21.DBB 476;
      T     DB22.DBB 8852;
_063: NOP   0;
      A     L 0.1;
      A(;
      L     DB20.DBW 62;
      L     14;
      ==I;
      );
      =     L 0.2;
      A     L 0.2;
      JNB   _064;
      L     DB21.DBW 6;
      T     DB22.DBW 8560;
_064: NOP   0;
      A     L 0.2;
      JNB   _065;
      L     DB21.DBW 8;
      T     DB22.DBW 8562;
_065: NOP   0;
      A     L 0.2;
      JNB   _066;
      L     DB21.DBB 476;
      T     DB22.DBB 8853;
_066: NOP   0;
      A     L 0.1;
      A(;
      L     DB20.DBW 62;
      L     15;
      ==I;
      );
      =     L 0.2;
      A     L 0.2;
      JNB   _067;
      L     DB21.DBW 6;
      T     DB22.DBW 8600;
_067: NOP   0;
      A     L 0.2;
      JNB   _068;
      L     DB21.DBW 8;
      T     DB22.DBW 8602;
_068: NOP   0;
      A     L 0.2;
      JNB   _069;
      L     DB21.DBB 476;
      T     DB22.DBB 8854;
_069: NOP   0;
      A     L 0.1;
      A(;
      L     DB20.DBW 62;
      L     16;
      ==I;
      );
      =     L 0.2;
      A     L 0.2;
      JNB   _06a;
      L     DB21.DBW 6;
      T     DB22.DBW 8640;
_06a: NOP   0;
      A     L 0.2;
      JNB   _06b;
      L     DB21.DBW 8;
      T     DB22.DBW 8642;
_06b: NOP   0;
      A     L 0.2;
      JNB   _06c;
      L     DB21.DBB 476;
      T     DB22.DBB 8855;
_06c: NOP   0;
      A     L 0.0;
      A     M 90.4;
      =     L 0.1;
      A     L 0.1;
      A(;
      L     DB20.DBW 62;
      L     17;
      ==I;
      );
      =     L 0.2;
      A     L 0.2;
      JNB   _06d;
      L     DB21.DBW 6;
      T     DB22.DBW 8680;
_06d: NOP   0;
      A     L 0.2;
      JNB   _06e;
      L     DB21.DBW 8;
      T     DB22.DBW 8682;
_06e: NOP   0;
      A     L 0.2;
      JNB   _06f;
      L     DB21.DBB 476;
      T     DB22.DBB 8856;
_06f: NOP   0;
      A     L 0.1;
      A(;
      L     DB20.DBW 62;
      L     18;
      ==I;
      );
      =     L 0.2;
      A     L 0.2;
      JNB   _070;
      L     DB21.DBW 6;
      T     DB22.DBW 8720;
_070: NOP   0;
      A     L 0.2;
      JNB   _071;
      L     DB21.DBW 8;
      T     DB22.DBW 8722;
_071: NOP   0;
      A     L 0.2;
      JNB   _072;
      L     DB21.DBB 476;
      T     DB22.DBB 8857;
_072: NOP   0;
      A     L 0.1;
      A(;
      L     DB20.DBW 62;
      L     19;
      ==I;
      );
      =     L 0.2;
      A     L 0.2;
      JNB   _073;
      L     DB21.DBW 6;
      T     DB22.DBW 8760;
_073: NOP   0;
      A     L 0.2;
      JNB   _074;
      L     DB21.DBW 8;
      T     DB22.DBW 8762;
_074: NOP   0;
      A     L 0.2;
      JNB   _075;
      L     DB21.DBB 476;
      T     DB22.DBB 8858;
_075: NOP   0;
      A     L 0.1;
      A(;
      L     DB20.DBW 62;
      L     20;
      ==I;
      );
      =     L 0.2;
      A     L 0.2;
      JNB   _076;
      L     DB21.DBW 6;
      T     DB22.DBW 8800;
_076: NOP   0;
      A     L 0.2;
      JNB   _077;
      L     DB21.DBW 8;
      T     DB22.DBW 8802;
_077: NOP   0;
      A     L 0.2;
      JNB   _078;
      L     DB21.DBB 476;
      T     DB22.DBB 8859;
_078: NOP   0;
NETWORK
TITLE =
NETWORK
TITLE =
      A     "On";
      =     L 0.0;
      A     L 0.0;
      A(;
      A(;
      L     DB21.DBW 370;
      L     0;
      ==I;
      );
      A     "AUT";
      O;
      A     "M11.2";
      A(;
      L     DB7.DBB 375;
      L     1;
      ==I;
      );
      A(;
      O(;
      L     DB7.DBW 2;
      L     5;
      ==I;
      );
      O(;
      L     DB7.DBW 2;
      L     11;
      ==I;
      );
      );
      );
      =     L 0.1;
      A(;
      A     L 0.1;
      A     DB21.DBX 394.0;
      JNB   _079;
      L     DB21.DBD 46;
      T     "MD588";
      SET;
      SAVE;
      CLR;
_079: A     BR;
      );
      JNB   _07a;
      L     DB21.DBD 50;
      T     "MD592";
_07a: NOP   0;
      A(;
      A     L 0.1;
      AN    DB21.DBX 394.0;
      JNB   _07b;
      L     DB21.DBD 54;
      T     "MD588";
      SET;
      SAVE;
      CLR;
_07b: A     BR;
      );
      JNB   _07c;
      L     DB21.DBD 58;
      T     "MD592";
_07c: NOP   0;
      A     L 0.0;
      A(;
      A(;
      L     DB21.DBW 370;
      L     1;
      ==I;
      );
      A     "AUT";
      O;
      A     "M11.2";
      A(;
      L     DB7.DBB 375;
      L     2;
      ==I;
      );
      A(;
      O(;
      L     DB7.DBW 2;
      L     5;
      ==I;
      );
      O(;
      L     DB7.DBW 2;
      L     11;
      ==I;
      );
      );
      );
      =     L 0.1;
      A(;
      A     L 0.1;
      A     DB21.DBX 394.0;
      JNB   _07d;
      L     DB21.DBD 62;
      T     "MD588";
      SET;
      SAVE;
      CLR;
_07d: A     BR;
      );
      JNB   _07e;
      L     DB21.DBD 66;
      T     "MD592";
_07e: NOP   0;
      A(;
      A     L 0.1;
      AN    DB21.DBX 394.0;
      JNB   _07f;
      L     DB21.DBD 70;
      T     "MD588";
      SET;
      SAVE;
      CLR;
_07f: A     BR;
      );
      JNB   _080;
      L     DB21.DBD 74;
      T     "MD592";
_080: NOP   0;
      A     L 0.0;
      A(;
      A(;
      L     DB21.DBW 370;
      L     2;
      ==I;
      );
      A     "AUT";
      O;
      A     "M11.2";
      A(;
      L     DB7.DBB 375;
      L     3;
      ==I;
      );
      A(;
      O(;
      L     DB7.DBW 2;
      L     5;
      ==I;
      );
      O(;
      L     DB7.DBW 2;
      L     11;
      ==I;
      );
      );
      );
      =     L 0.1;
      A(;
      A     L 0.1;
      A     DB21.DBX 394.0;
      JNB   _081;
      L     DB21.DBD 78;
      T     "MD588";
      SET;
      SAVE;
      CLR;
_081: A     BR;
      );
      JNB   _082;
      L     DB21.DBD 82;
      T     "MD592";
_082: NOP   0;
      A(;
      A     L 0.1;
      AN    DB21.DBX 394.0;
      JNB   _083;
      L     DB21.DBD 86;
      T     "MD588";
      SET;
      SAVE;
      CLR;
_083: A     BR;
      );
      JNB   _084;
      L     DB21.DBD 90;
      T     "MD592";
_084: NOP   0;
      A     L 0.0;
      A(;
      A(;
      L     DB21.DBW 370;
      L     3;
      ==I;
      );
      A     "AUT";
      O;
      A     "M11.2";
      A(;
      L     DB7.DBB 375;
      L     4;
      ==I;
      );
      A(;
      O(;
      L     DB7.DBW 2;
      L     5;
      ==I;
      );
      O(;
      L     DB7.DBW 2;
      L     11;
      ==I;
      );
      );
      );
      =     L 0.1;
      A(;
      A     L 0.1;
      A     DB21.DBX 394.0;
      JNB   _085;
      L     DB21.DBD 94;
      T     "MD588";
      SET;
      SAVE;
      CLR;
_085: A     BR;
      );
      JNB   _086;
      L     DB21.DBD 98;
      T     "MD592";
_086: NOP   0;
      A(;
      A     L 0.1;
      AN    DB21.DBX 394.0;
      JNB   _087;
      L     DB21.DBD 102;
      T     "MD588";
      SET;
      SAVE;
      CLR;
_087: A     BR;
      );
      JNB   _088;
      L     DB21.DBD 106;
      T     "MD592";
_088: NOP   0;
      A     L 0.0;
      A(;
      A(;
      L     DB21.DBW 370;
      L     4;
      ==I;
      );
      A     "AUT";
      O;
      A     "M11.2";
      A(;
      L     DB7.DBB 375;
      L     5;
      ==I;
      );
      A(;
      O(;
      L     DB7.DBW 2;
      L     5;
      ==I;
      );
      O(;
      L     DB7.DBW 2;
      L     11;
      ==I;
      );
      );
      );
      =     L 0.1;
      A(;
      A     L 0.1;
      A     DB21.DBX 394.0;
      JNB   _089;
      L     DB21.DBD 110;
      T     "MD588";
      SET;
      SAVE;
      CLR;
_089: A     BR;
      );
      JNB   _08a;
      L     DB21.DBD 114;
      T     "MD592";
_08a: NOP   0;
      A(;
      A     L 0.1;
      AN    DB21.DBX 394.0;
      JNB   _08b;
      L     DB21.DBD 118;
      T     "MD588";
      SET;
      SAVE;
      CLR;
_08b: A     BR;
      );
      JNB   _08c;
      L     DB21.DBD 122;
      T     "MD592";
_08c: NOP   0;
      A     L 0.0;
      A(;
      A(;
      L     DB21.DBW 370;
      L     5;
      ==I;
      );
      A     "AUT";
      O;
      A     "M11.2";
      A(;
      L     DB7.DBB 375;
      L     6;
      ==I;
      );
      A(;
      O(;
      L     DB7.DBW 2;
      L     5;
      ==I;
      );
      O(;
      L     DB7.DBW 2;
      L     11;
      ==I;
      );
      );
      );
      =     L 0.1;
      A(;
      A     L 0.1;
      A     DB21.DBX 394.0;
      JNB   _08d;
      L     DB21.DBD 126;
      T     "MD588";
      SET;
      SAVE;
      CLR;
_08d: A     BR;
      );
      JNB   _08e;
      L     DB21.DBD 130;
      T     "MD592";
_08e: NOP   0;
      A(;
      A     L 0.1;
      AN    DB21.DBX 394.0;
      JNB   _08f;
      L     DB21.DBD 134;
      T     "MD588";
      SET;
      SAVE;
      CLR;
_08f: A     BR;
      );
      JNB   _090;
      L     DB21.DBD 138;
      T     "MD592";
_090: NOP   0;
      A     L 0.0;
      A(;
      A(;
      L     DB21.DBW 370;
      L     6;
      ==I;
      );
      A     "AUT";
      O;
      A     "M11.2";
      A(;
      L     DB7.DBB 375;
      L     7;
      ==I;
      );
      A(;
      O(;
      L     DB7.DBW 2;
      L     5;
      ==I;
      );
      O(;
      L     DB7.DBW 2;
      L     11;
      ==I;
      );
      );
      );
      =     L 0.1;
      A(;
      A     L 0.1;
      A     DB21.DBX 394.0;
      JNB   _091;
      L     DB21.DBD 142;
      T     "MD588";
      SET;
      SAVE;
      CLR;
_091: A     BR;
      );
      JNB   _092;
      L     DB21.DBD 146;
      T     "MD592";
_092: NOP   0;
      A(;
      A     L 0.1;
      AN    DB21.DBX 394.0;
      JNB   _093;
      L     DB21.DBD 150;
      T     "MD588";
      SET;
      SAVE;
      CLR;
_093: A     BR;
      );
      JNB   _094;
      L     DB21.DBD 154;
      T     "MD592";
_094: NOP   0;
      A     L 0.0;
      A(;
      A(;
      L     DB21.DBW 370;
      L     7;
      ==I;
      );
      A     "AUT";
      O;
      A     "M11.2";
      A(;
      L     DB7.DBB 375;
      L     8;
      ==I;
      );
      A(;
      O(;
      L     DB7.DBW 2;
      L     5;
      ==I;
      );
      O(;
      L     DB7.DBW 2;
      L     11;
      ==I;
      );
      );
      );
      =     L 0.1;
      A(;
      A     L 0.1;
      A     DB21.DBX 394.0;
      JNB   _095;
      L     DB21.DBD 158;
      T     "MD588";
      SET;
      SAVE;
      CLR;
_095: A     BR;
      );
      JNB   _096;
      L     DB21.DBD 162;
      T     "MD592";
_096: NOP   0;
      A(;
      A     L 0.1;
      AN    DB21.DBX 394.0;
      JNB   _097;
      L     DB21.DBD 166;
      T     "MD588";
      SET;
      SAVE;
      CLR;
_097: A     BR;
      );
      JNB   _098;
      L     DB21.DBD 170;
      T     "MD592";
_098: NOP   0;
      A     L 0.0;
      A(;
      A(;
      L     DB21.DBW 370;
      L     8;
      ==I;
      );
      A     "AUT";
      O;
      A     "M11.2";
      A(;
      L     DB7.DBB 375;
      L     9;
      ==I;
      );
      A(;
      O(;
      L     DB7.DBW 2;
      L     5;
      ==I;
      );
      O(;
      L     DB7.DBW 2;
      L     11;
      ==I;
      );
      );
      );
      =     L 0.1;
      A(;
      A     L 0.1;
      A     DB21.DBX 394.0;
      JNB   _099;
      L     DB21.DBD 174;
      T     "MD588";
      SET;
      SAVE;
      CLR;
_099: A     BR;
      );
      JNB   _09a;
      L     DB21.DBD 178;
      T     "MD592";
_09a: NOP   0;
      A(;
      A     L 0.1;
      AN    DB21.DBX 394.0;
      JNB   _09b;
      L     DB21.DBD 182;
      T     "MD588";
      SET;
      SAVE;
      CLR;
_09b: A     BR;
      );
      JNB   _09c;
      L     DB21.DBD 186;
      T     "MD592";
_09c: NOP   0;
      A     L 0.0;
      A(;
      A(;
      L     DB21.DBW 370;
      L     9;
      ==I;
      );
      A     "AUT";
      O;
      A     "M11.2";
      A(;
      L     DB7.DBB 375;
      L     10;
      ==I;
      );
      A(;
      O(;
      L     DB7.DBW 2;
      L     5;
      ==I;
      );
      O(;
      L     DB7.DBW 2;
      L     11;
      ==I;
      );
      );
      );
      =     L 0.1;
      A(;
      A     L 0.1;
      A     DB21.DBX 394.0;
      JNB   _09d;
      L     DB21.DBD 190;
      T     "MD588";
      SET;
      SAVE;
      CLR;
_09d: A     BR;
      );
      JNB   _09e;
      L     DB21.DBD 194;
      T     "MD592";
_09e: NOP   0;
      A(;
      A     L 0.1;
      AN    DB21.DBX 394.0;
      JNB   _09f;
      L     DB21.DBD 198;
      T     "MD588";
      SET;
      SAVE;
      CLR;
_09f: A     BR;
      );
      JNB   _0a0;
      L     DB21.DBD 202;
      T     "MD592";
_0a0: NOP   0;
      A     L 0.0;
      A(;
      A(;
      L     DB21.DBW 370;
      L     10;
      ==I;
      );
      A     "AUT";
      O;
      A     "M11.2";
      A(;
      L     DB7.DBB 375;
      L     11;
      ==I;
      );
      A(;
      O(;
      L     DB7.DBW 2;
      L     5;
      ==I;
      );
      O(;
      L     DB7.DBW 2;
      L     11;
      ==I;
      );
      );
      );
      =     L 0.1;
      A(;
      A     L 0.1;
      A     DB21.DBX 394.0;
      JNB   _0a1;
      L     DB21.DBD 206;
      T     "MD588";
      SET;
      SAVE;
      CLR;
_0a1: A     BR;
      );
      JNB   _0a2;
      L     DB21.DBD 210;
      T     "MD592";
_0a2: NOP   0;
      A(;
      A     L 0.1;
      AN    DB21.DBX 394.0;
      JNB   _0a3;
      L     DB21.DBD 214;
      T     "MD588";
      SET;
      SAVE;
      CLR;
_0a3: A     BR;
      );
      JNB   _0a4;
      L     DB21.DBD 218;
      T     "MD592";
_0a4: NOP   0;
      A     L 0.0;
      A(;
      A(;
      L     DB21.DBW 370;
      L     11;
      ==I;
      );
      A     "AUT";
      O;
      A     "M11.2";
      A(;
      L     DB7.DBB 375;
      L     12;
      ==I;
      );
      A(;
      O(;
      L     DB7.DBW 2;
      L     5;
      ==I;
      );
      O(;
      L     DB7.DBW 2;
      L     11;
      ==I;
      );
      );
      );
      =     L 0.1;
      A(;
      A     L 0.1;
      A     DB21.DBX 394.0;
      JNB   _0a5;
      L     DB21.DBD 222;
      T     "MD588";
      SET;
      SAVE;
      CLR;
_0a5: A     BR;
      );
      JNB   _0a6;
      L     DB21.DBD 226;
      T     "MD592";
_0a6: NOP   0;
      A(;
      A     L 0.1;
      AN    DB21.DBX 394.0;
      JNB   _0a7;
      L     DB21.DBD 230;
      T     "MD588";
      SET;
      SAVE;
      CLR;
_0a7: A     BR;
      );
      JNB   _0a8;
      L     DB21.DBD 234;
      T     "MD592";
_0a8: NOP   0;
      A     L 0.0;
      A(;
      A(;
      L     DB21.DBW 370;
      L     12;
      ==I;
      );
      A     "AUT";
      O;
      A     "M11.2";
      A(;
      L     DB7.DBB 375;
      L     13;
      ==I;
      );
      A(;
      O(;
      L     DB7.DBW 2;
      L     5;
      ==I;
      );
      O(;
      L     DB7.DBW 2;
      L     11;
      ==I;
      );
      );
      );
      =     L 0.1;
      A(;
      A     L 0.1;
      A     DB21.DBX 394.0;
      JNB   _0a9;
      L     DB21.DBD 238;
      T     "MD588";
      SET;
      SAVE;
      CLR;
_0a9: A     BR;
      );
      JNB   _0aa;
      L     DB21.DBD 242;
      T     "MD592";
_0aa: NOP   0;
      A(;
      A     L 0.1;
      AN    DB21.DBX 394.0;
      JNB   _0ab;
      L     DB21.DBD 246;
      T     "MD588";
      SET;
      SAVE;
      CLR;
_0ab: A     BR;
      );
      JNB   _0ac;
      L     DB21.DBD 250;
      T     "MD592";
_0ac: NOP   0;
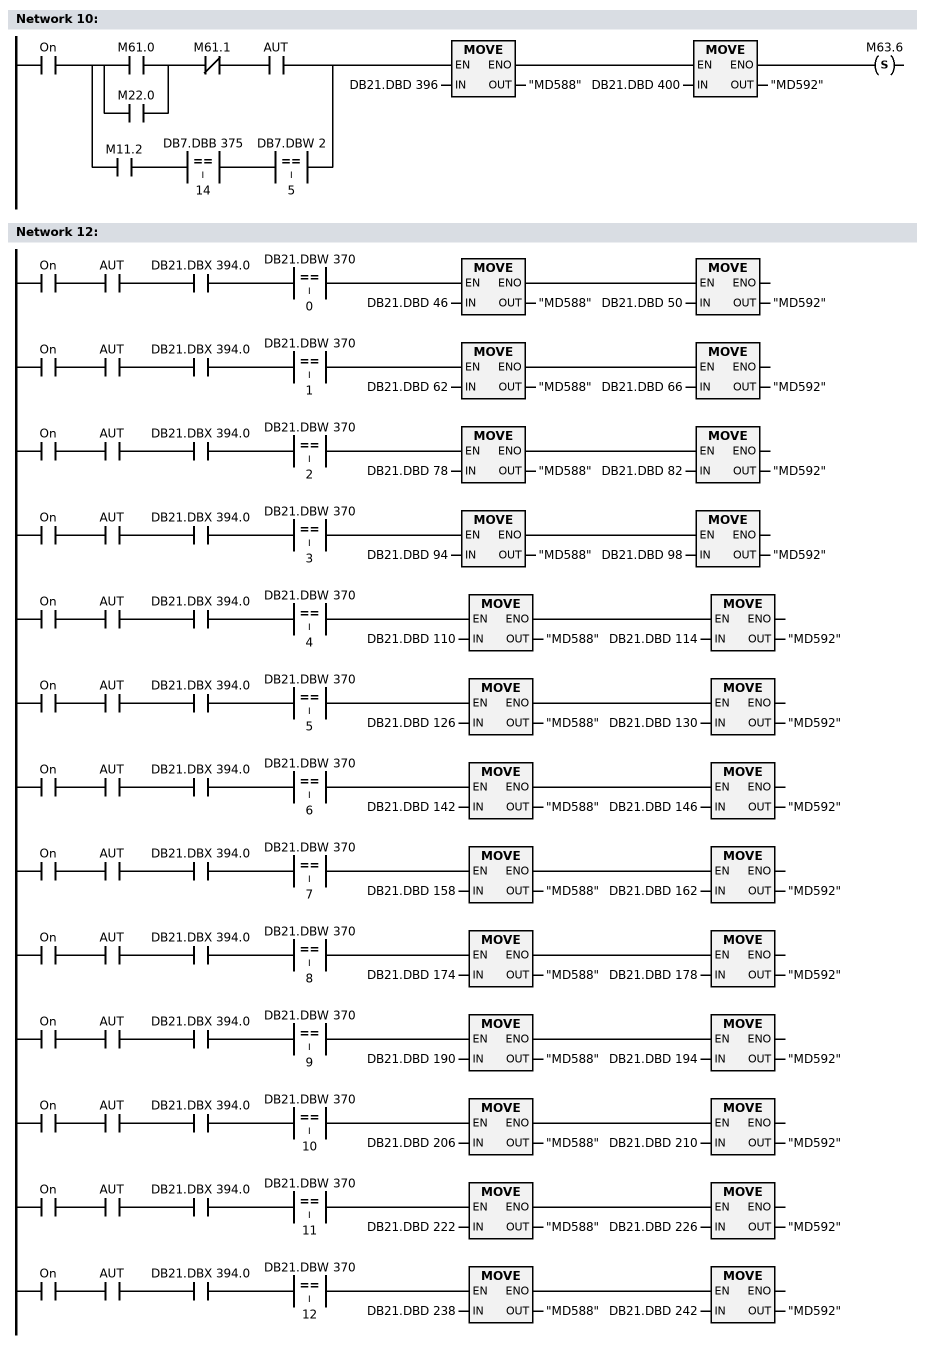
NETWORK
TITLE =
      A(;
      A     "On";
      A(;
      A(;
      O     "M61.0";
      O     "M22.0";
      );
      AN    "M61.1";
      A     "AUT";
      O;
      A     "M11.2";
      A(;
      L     DB7.DBB 375;
      L     14;
      ==I;
      );
      A(;
      L     DB7.DBW 2;
      L     5;
      ==I;
      );
      );
      JNB   _0ad;
      L     DB21.DBD 396;
      T     "MD588";
      SET;
      SAVE;
      CLR;
_0ad: A     BR;
      );
      JNB   _0ae;
      L     DB21.DBD 400;
      T     "MD592";
      SET;
      SAVE;
      CLR;
_0ae: A     BR;
      S     "M63.6";
NETWORK
TITLE =
NETWORK
TITLE =
      A     "On";
      A     "AUT";
      A     DB21.DBX 394.0;
      =     L 0.0;
      A(;
      A     L 0.0;
      A(;
      L     DB21.DBW 370;
      L     0;
      ==I;
      );
      JNB   _0af;
      L     DB21.DBD 46;
      T     "MD588";
      SET;
      SAVE;
      CLR;
_0af: A     BR;
      );
      JNB   _0b0;
      L     DB21.DBD 50;
      T     "MD592";
_0b0: NOP   0;
      A(;
      A     L 0.0;
      A(;
      L     DB21.DBW 370;
      L     1;
      ==I;
      );
      JNB   _0b1;
      L     DB21.DBD 62;
      T     "MD588";
      SET;
      SAVE;
      CLR;
_0b1: A     BR;
      );
      JNB   _0b2;
      L     DB21.DBD 66;
      T     "MD592";
_0b2: NOP   0;
      A(;
      A     L 0.0;
      A(;
      L     DB21.DBW 370;
      L     2;
      ==I;
      );
      JNB   _0b3;
      L     DB21.DBD 78;
      T     "MD588";
      SET;
      SAVE;
      CLR;
_0b3: A     BR;
      );
      JNB   _0b4;
      L     DB21.DBD 82;
      T     "MD592";
_0b4: NOP   0;
      A(;
      A     L 0.0;
      A(;
      L     DB21.DBW 370;
      L     3;
      ==I;
      );
      JNB   _0b5;
      L     DB21.DBD 94;
      T     "MD588";
      SET;
      SAVE;
      CLR;
_0b5: A     BR;
      );
      JNB   _0b6;
      L     DB21.DBD 98;
      T     "MD592";
_0b6: NOP   0;
      A(;
      A     L 0.0;
      A(;
      L     DB21.DBW 370;
      L     4;
      ==I;
      );
      JNB   _0b7;
      L     DB21.DBD 110;
      T     "MD588";
      SET;
      SAVE;
      CLR;
_0b7: A     BR;
      );
      JNB   _0b8;
      L     DB21.DBD 114;
      T     "MD592";
_0b8: NOP   0;
      A(;
      A     L 0.0;
      A(;
      L     DB21.DBW 370;
      L     5;
      ==I;
      );
      JNB   _0b9;
      L     DB21.DBD 126;
      T     "MD588";
      SET;
      SAVE;
      CLR;
_0b9: A     BR;
      );
      JNB   _0ba;
      L     DB21.DBD 130;
      T     "MD592";
_0ba: NOP   0;
      A(;
      A     L 0.0;
      A(;
      L     DB21.DBW 370;
      L     6;
      ==I;
      );
      JNB   _0bb;
      L     DB21.DBD 142;
      T     "MD588";
      SET;
      SAVE;
      CLR;
_0bb: A     BR;
      );
      JNB   _0bc;
      L     DB21.DBD 146;
      T     "MD592";
_0bc: NOP   0;
      A(;
      A     L 0.0;
      A(;
      L     DB21.DBW 370;
      L     7;
      ==I;
      );
      JNB   _0bd;
      L     DB21.DBD 158;
      T     "MD588";
      SET;
      SAVE;
      CLR;
_0bd: A     BR;
      );
      JNB   _0be;
      L     DB21.DBD 162;
      T     "MD592";
_0be: NOP   0;
      A(;
      A     L 0.0;
      A(;
      L     DB21.DBW 370;
      L     8;
      ==I;
      );
      JNB   _0bf;
      L     DB21.DBD 174;
      T     "MD588";
      SET;
      SAVE;
      CLR;
_0bf: A     BR;
      );
      JNB   _0c0;
      L     DB21.DBD 178;
      T     "MD592";
_0c0: NOP   0;
      A(;
      A     L 0.0;
      A(;
      L     DB21.DBW 370;
      L     9;
      ==I;
      );
      JNB   _0c1;
      L     DB21.DBD 190;
      T     "MD588";
      SET;
      SAVE;
      CLR;
_0c1: A     BR;
      );
      JNB   _0c2;
      L     DB21.DBD 194;
      T     "MD592";
_0c2: NOP   0;
      A(;
      A     L 0.0;
      A(;
      L     DB21.DBW 370;
      L     10;
      ==I;
      );
      JNB   _0c3;
      L     DB21.DBD 206;
      T     "MD588";
      SET;
      SAVE;
      CLR;
_0c3: A     BR;
      );
      JNB   _0c4;
      L     DB21.DBD 210;
      T     "MD592";
_0c4: NOP   0;
      A(;
      A     L 0.0;
      A(;
      L     DB21.DBW 370;
      L     11;
      ==I;
      );
      JNB   _0c5;
      L     DB21.DBD 222;
      T     "MD588";
      SET;
      SAVE;
      CLR;
_0c5: A     BR;
      );
      JNB   _0c6;
      L     DB21.DBD 226;
      T     "MD592";
_0c6: NOP   0;
      A(;
      A     L 0.0;
      A(;
      L     DB21.DBW 370;
      L     12;
      ==I;
      );
      JNB   _0c7;
      L     DB21.DBD 238;
      T     "MD588";
      SET;
      SAVE;
      CLR;
_0c7: A     BR;
      );
      JNB   _0c8;
      L     DB21.DBD 242;
      T     "MD592";
_0c8: NOP   0;
NETWORK
TITLE =
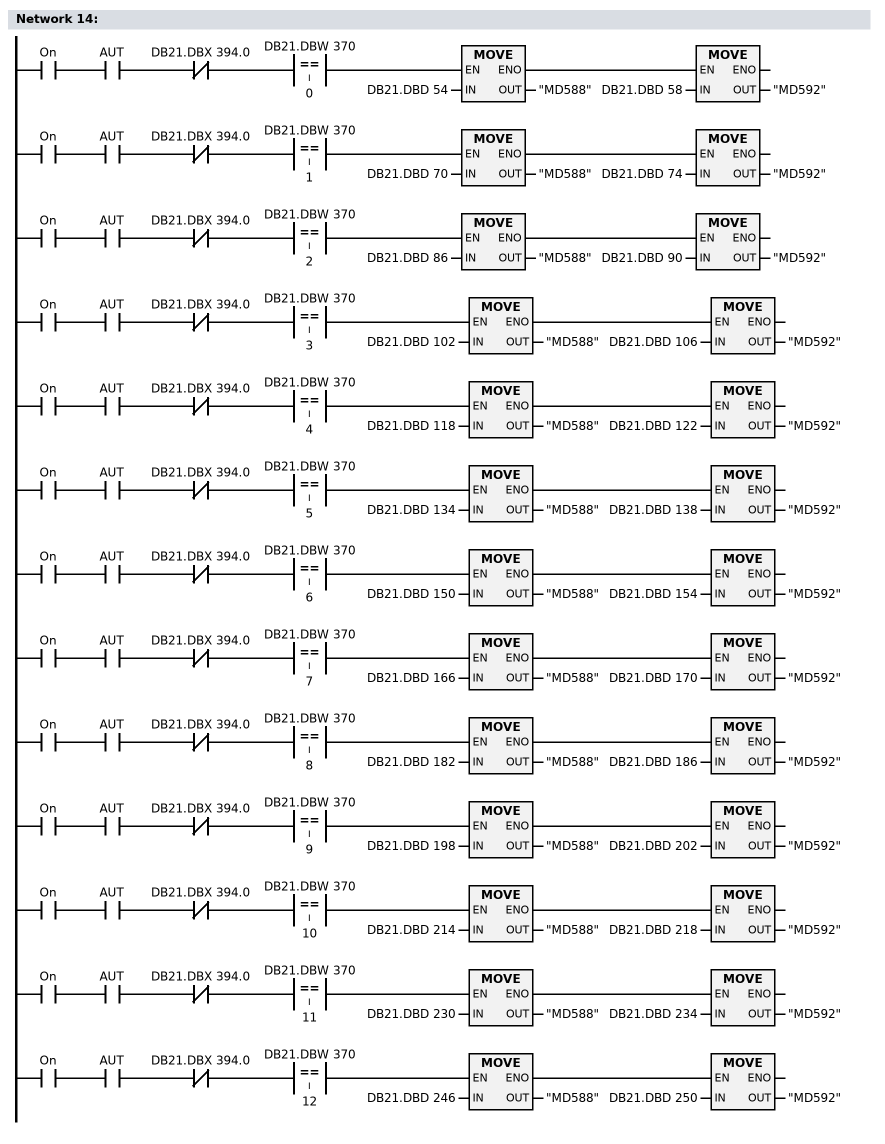
NETWORK
TITLE =
      A     "On";
      A     "AUT";
      AN    DB21.DBX 394.0;
      =     L 0.0;
      A(;
      A     L 0.0;
      A(;
      L     DB21.DBW 370;
      L     0;
      ==I;
      );
      JNB   _0c9;
      L     DB21.DBD 54;
      T     "MD588";
      SET;
      SAVE;
      CLR;
_0c9: A     BR;
      );
      JNB   _0ca;
      L     DB21.DBD 58;
      T     "MD592";
_0ca: NOP   0;
      A(;
      A     L 0.0;
      A(;
      L     DB21.DBW 370;
      L     1;
      ==I;
      );
      JNB   _0cb;
      L     DB21.DBD 70;
      T     "MD588";
      SET;
      SAVE;
      CLR;
_0cb: A     BR;
      );
      JNB   _0cc;
      L     DB21.DBD 74;
      T     "MD592";
_0cc: NOP   0;
      A(;
      A     L 0.0;
      A(;
      L     DB21.DBW 370;
      L     2;
      ==I;
      );
      JNB   _0cd;
      L     DB21.DBD 86;
      T     "MD588";
      SET;
      SAVE;
      CLR;
_0cd: A     BR;
      );
      JNB   _0ce;
      L     DB21.DBD 90;
      T     "MD592";
_0ce: NOP   0;
      A(;
      A     L 0.0;
      A(;
      L     DB21.DBW 370;
      L     3;
      ==I;
      );
      JNB   _0cf;
      L     DB21.DBD 102;
      T     "MD588";
      SET;
      SAVE;
      CLR;
_0cf: A     BR;
      );
      JNB   _0d0;
      L     DB21.DBD 106;
      T     "MD592";
_0d0: NOP   0;
      A(;
      A     L 0.0;
      A(;
      L     DB21.DBW 370;
      L     4;
      ==I;
      );
      JNB   _0d1;
      L     DB21.DBD 118;
      T     "MD588";
      SET;
      SAVE;
      CLR;
_0d1: A     BR;
      );
      JNB   _0d2;
      L     DB21.DBD 122;
      T     "MD592";
_0d2: NOP   0;
      A(;
      A     L 0.0;
      A(;
      L     DB21.DBW 370;
      L     5;
      ==I;
      );
      JNB   _0d3;
      L     DB21.DBD 134;
      T     "MD588";
      SET;
      SAVE;
      CLR;
_0d3: A     BR;
      );
      JNB   _0d4;
      L     DB21.DBD 138;
      T     "MD592";
_0d4: NOP   0;
      A(;
      A     L 0.0;
      A(;
      L     DB21.DBW 370;
      L     6;
      ==I;
      );
      JNB   _0d5;
      L     DB21.DBD 150;
      T     "MD588";
      SET;
      SAVE;
      CLR;
_0d5: A     BR;
      );
      JNB   _0d6;
      L     DB21.DBD 154;
      T     "MD592";
_0d6: NOP   0;
      A(;
      A     L 0.0;
      A(;
      L     DB21.DBW 370;
      L     7;
      ==I;
      );
      JNB   _0d7;
      L     DB21.DBD 166;
      T     "MD588";
      SET;
      SAVE;
      CLR;
_0d7: A     BR;
      );
      JNB   _0d8;
      L     DB21.DBD 170;
      T     "MD592";
_0d8: NOP   0;
      A(;
      A     L 0.0;
      A(;
      L     DB21.DBW 370;
      L     8;
      ==I;
      );
      JNB   _0d9;
      L     DB21.DBD 182;
      T     "MD588";
      SET;
      SAVE;
      CLR;
_0d9: A     BR;
      );
      JNB   _0da;
      L     DB21.DBD 186;
      T     "MD592";
_0da: NOP   0;
      A(;
      A     L 0.0;
      A(;
      L     DB21.DBW 370;
      L     9;
      ==I;
      );
      JNB   _0db;
      L     DB21.DBD 198;
      T     "MD588";
      SET;
      SAVE;
      CLR;
_0db: A     BR;
      );
      JNB   _0dc;
      L     DB21.DBD 202;
      T     "MD592";
_0dc: NOP   0;
      A(;
      A     L 0.0;
      A(;
      L     DB21.DBW 370;
      L     10;
      ==I;
      );
      JNB   _0dd;
      L     DB21.DBD 214;
      T     "MD588";
      SET;
      SAVE;
      CLR;
_0dd: A     BR;
      );
      JNB   _0de;
      L     DB21.DBD 218;
      T     "MD592";
_0de: NOP   0;
      A(;
      A     L 0.0;
      A(;
      L     DB21.DBW 370;
      L     11;
      ==I;
      );
      JNB   _0df;
      L     DB21.DBD 230;
      T     "MD588";
      SET;
      SAVE;
      CLR;
_0df: A     BR;
      );
      JNB   _0e0;
      L     DB21.DBD 234;
      T     "MD592";
_0e0: NOP   0;
      A(;
      A     L 0.0;
      A(;
      L     DB21.DBW 370;
      L     12;
      ==I;
      );
      JNB   _0e1;
      L     DB21.DBD 246;
      T     "MD588";
      SET;
      SAVE;
      CLR;
_0e1: A     BR;
      );
      JNB   _0e2;
      L     DB21.DBD 250;
      T     "MD592";
_0e2: NOP   0;
NETWORK
TITLE =
END_FUNCTION

FUNCTION "FC81 - GEST AXIS" : VOID	// FC 81
VERSION : 0.1
BEGIN
// (block stored without names or comments; labels and parameter names are numbered)
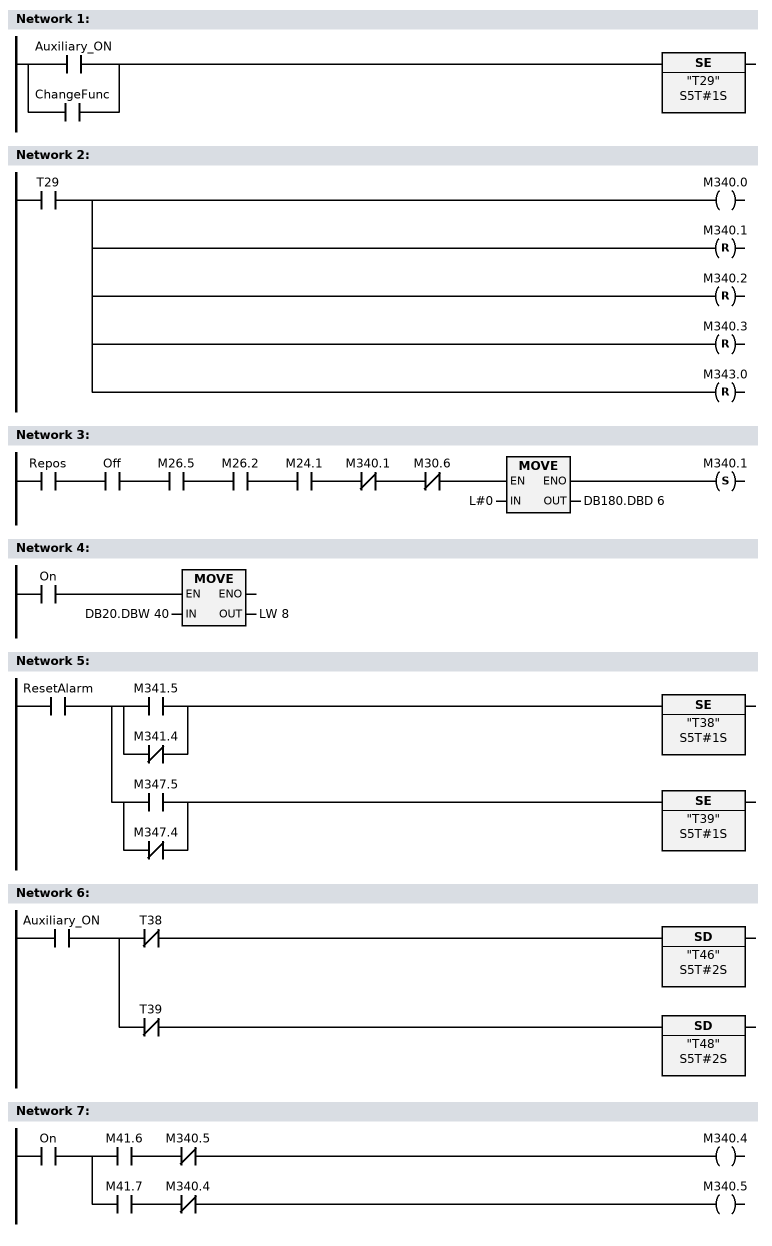
NETWORK
TITLE =
      O     "Auxiliary_ON";
      O     "ChangeFunc";
      L     S5T#1S;
      SE    "T29";
NETWORK
TITLE =
      A     "T29";
      =     "M340.0";
      R     "M340.1";
      R     "M340.2";
      R     "M340.3";
      R     "M343.0";
NETWORK
TITLE =
      A     "Repos";
      A     "Off";
      A     "M26.5";
      A     "M26.2";
      A     "M24.1";
      AN    "M340.1";
      AN    "M30.6";
      JNB   M001;
      L     L#0;
      T     DB180.DBD 6;
      SET;
      SAVE;
      CLR;
M001: A     BR;
      S     "M340.1";
NETWORK
TITLE =
      A     "On";
      JNB   M002;
      L     DB20.DBW 40;
      T     LW 8;
M002: NOP   0;
NETWORK
TITLE =
      A     "ResetAlarm";
      =     L 15.0;
      A     L 15.0;
      A(;
      O     "M341.5";
      ON    "M341.4";
      );
      L     S5T#1S;
      SE    "T38";
      A     L 15.0;
      A(;
      O     "M347.5";
      ON    "M347.4";
      );
      L     S5T#1S;
      SE    "T39";
NETWORK
TITLE =
      A     "Auxiliary_ON";
      =     L 15.0;
      A     L 15.0;
      AN    "T38";
      L     S5T#2S;
      SD    "T46";
      A     L 15.0;
      AN    "T39";
      L     S5T#2S;
      SD    "T48";
NETWORK
TITLE =
      A     "On";
      =     L 15.0;
      A     L 15.0;
      A     "M41.6";
      AN    "M340.5";
      =     "M340.4";
      A     L 15.0;
      A     "M41.7";
      AN    "M340.4";
      =     "M340.5";
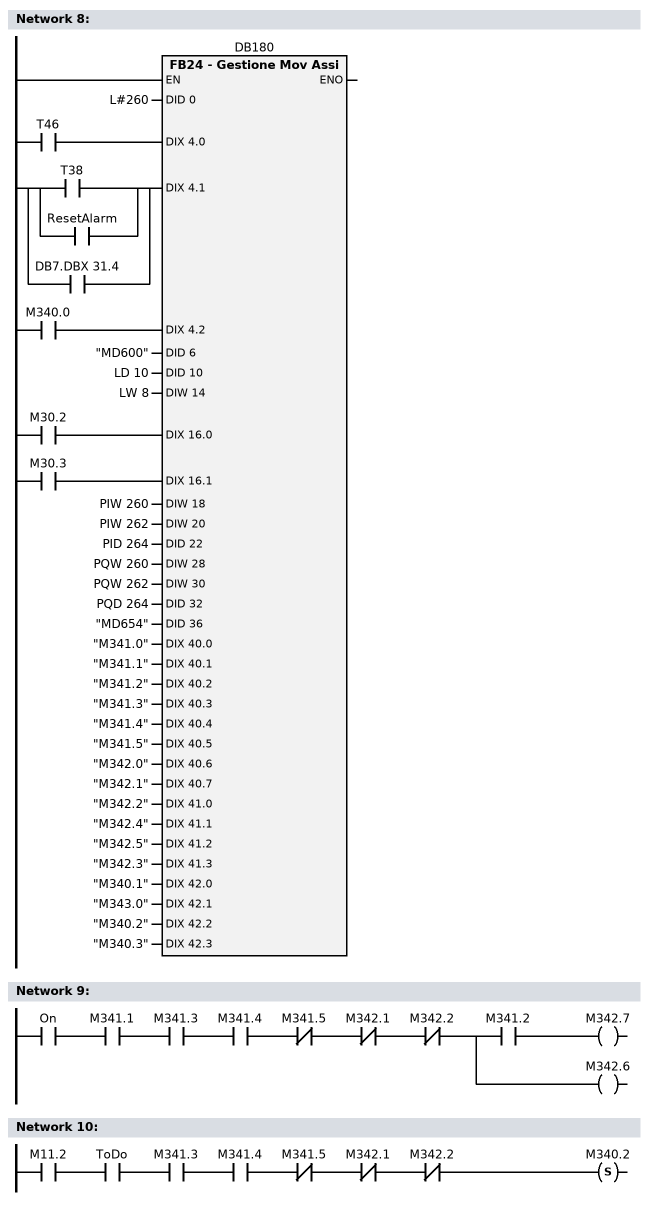
NETWORK
TITLE =
      A     "T46";
      =     L 15.0;
      BLD   103;
      A(;
      O     "T38";
      O     "ResetAlarm";
      O     DB7.DBX 31.4;
      );
      =     L 15.1;
      BLD   103;
      A     "M340.0";
      =     L 15.2;
      BLD   103;
      A     "M30.2";
      =     L 15.3;
      BLD   103;
      A     "M30.3";
      =     L 15.4;
      BLD   103;
      CALL  "FB24 - Gestione Mov Assi" , "DB180" (
           DID 0                    := L#260,
           DIX 4.0                  := L 15.0,
           DIX 4.1                  := L 15.1,
           DIX 4.2                  := L 15.2,
           DID 6                    := "MD600",
           DID 10                   := LD 10,
           DIW 14                   := LW 8,
           DIX 16.0                 := L 15.3,
           DIX 16.1                 := L 15.4,
           DIW 18                   := PIW 260,
           DIW 20                   := PIW 262,
           DID 22                   := PID 264,
           DIW 28                   := PQW 260,
           DIW 30                   := PQW 262,
           DID 32                   := PQD 264,
           DID 36                   := "MD654",
           DIX 40.0                 := "M341.0",
           DIX 40.1                 := "M341.1",
           DIX 40.2                 := "M341.2",
           DIX 40.3                 := "M341.3",
           DIX 40.4                 := "M341.4",
           DIX 40.5                 := "M341.5",
           DIX 40.6                 := "M342.0",
           DIX 40.7                 := "M342.1",
           DIX 41.0                 := "M342.2",
           DIX 41.1                 := "M342.4",
           DIX 41.2                 := "M342.5",
           DIX 41.3                 := "M342.3",
           DIX 42.0                 := "M340.1",
           DIX 42.1                 := "M343.0",
           DIX 42.2                 := "M340.2",
           DIX 42.3                 := "M340.3");
      NOP   0;
NETWORK
TITLE =
      A     "On";
      A     "M341.1";
      A     "M341.3";
      A     "M341.4";
      AN    "M341.5";
      AN    "M342.1";
      AN    "M342.2";
      =     L 15.0;
      A     L 15.0;
      A     "M341.2";
      =     "M342.7";
      A     L 15.0;
      BLD   102;
      =     "M342.6";
NETWORK
TITLE =
      A     "M11.2";
      A     "ToDo";
      A     "M341.3";
      A     "M341.4";
      AN    "M341.5";
      AN    "M342.1";
      AN    "M342.2";
      S     "M340.2";
NETWORK
TITLE =
NETWORK
TITLE =
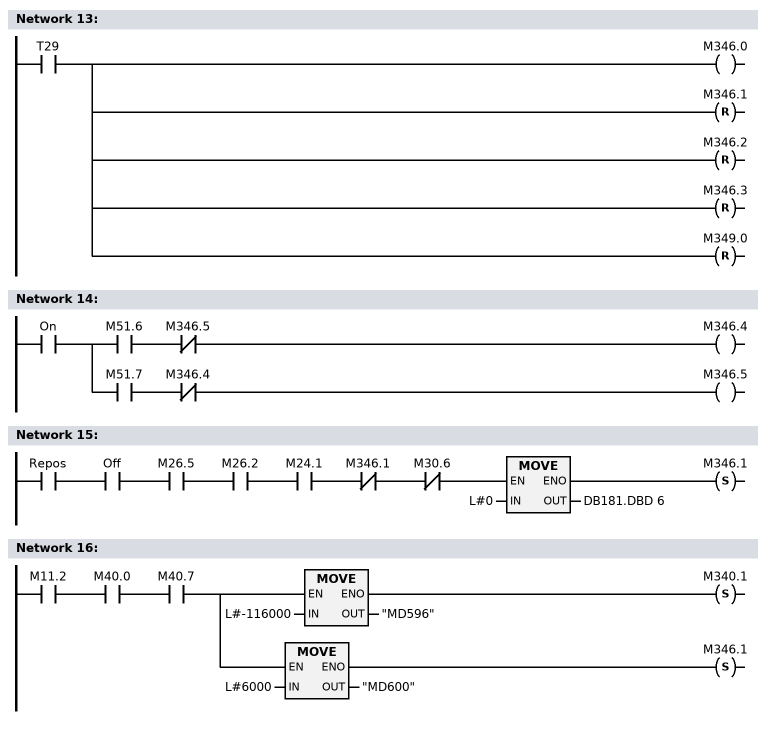
NETWORK
TITLE =
      A     "T29";
      =     "M346.0";
      R     "M346.1";
      R     "M346.2";
      R     "M346.3";
      R     "M349.0";
NETWORK
TITLE =
      A     "On";
      =     L 15.0;
      A     L 15.0;
      A     "M51.6";
      AN    "M346.5";
      =     "M346.4";
      A     L 15.0;
      A     "M51.7";
      AN    "M346.4";
      =     "M346.5";
NETWORK
TITLE =
      A     "Repos";
      A     "Off";
      A     "M26.5";
      A     "M26.2";
      A     "M24.1";
      AN    "M346.1";
      AN    "M30.6";
      JNB   M003;
      L     L#0;
      T     DB181.DBD 6;
      SET;
      SAVE;
      CLR;
M003: A     BR;
      S     "M346.1";
NETWORK
TITLE =
      A     "M11.2";
      A     "M40.0";
      A     "M40.7";
      =     L 15.0;
      A     L 15.0;
      JNB   M004;
      L     L#-116000;
      T     "MD596";
      SET;
      SAVE;
      CLR;
M004: A     BR;
      S     "M340.1";
      A     L 15.0;
      JNB   M005;
      L     L#6000;
      T     "MD600";
      SET;
      SAVE;
      CLR;
M005: A     BR;
      S     "M346.1";
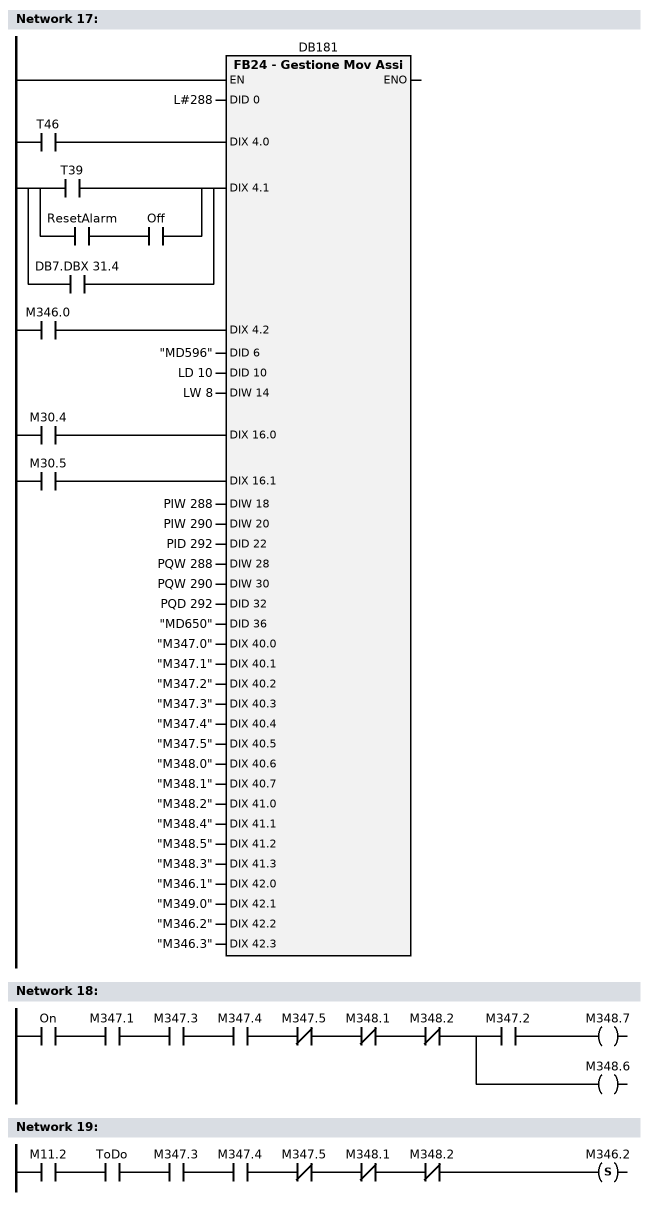
NETWORK
TITLE =
      A     "T46";
      =     L 15.0;
      BLD   103;
      A(;
      O     "T39";
      O;
      A     "ResetAlarm";
      A     "Off";
      O     DB7.DBX 31.4;
      );
      =     L 15.1;
      BLD   103;
      A     "M346.0";
      =     L 15.2;
      BLD   103;
      A     "M30.4";
      =     L 15.3;
      BLD   103;
      A     "M30.5";
      =     L 15.4;
      BLD   103;
      CALL  "FB24 - Gestione Mov Assi" , "DB181" (
           DID 0                    := L#288,
           DIX 4.0                  := L 15.0,
           DIX 4.1                  := L 15.1,
           DIX 4.2                  := L 15.2,
           DID 6                    := "MD596",
           DID 10                   := LD 10,
           DIW 14                   := LW 8,
           DIX 16.0                 := L 15.3,
           DIX 16.1                 := L 15.4,
           DIW 18                   := PIW 288,
           DIW 20                   := PIW 290,
           DID 22                   := PID 292,
           DIW 28                   := PQW 288,
           DIW 30                   := PQW 290,
           DID 32                   := PQD 292,
           DID 36                   := "MD650",
           DIX 40.0                 := "M347.0",
           DIX 40.1                 := "M347.1",
           DIX 40.2                 := "M347.2",
           DIX 40.3                 := "M347.3",
           DIX 40.4                 := "M347.4",
           DIX 40.5                 := "M347.5",
           DIX 40.6                 := "M348.0",
           DIX 40.7                 := "M348.1",
           DIX 41.0                 := "M348.2",
           DIX 41.1                 := "M348.4",
           DIX 41.2                 := "M348.5",
           DIX 41.3                 := "M348.3",
           DIX 42.0                 := "M346.1",
           DIX 42.1                 := "M349.0",
           DIX 42.2                 := "M346.2",
           DIX 42.3                 := "M346.3");
      NOP   0;
NETWORK
TITLE =
      A     "On";
      A     "M347.1";
      A     "M347.3";
      A     "M347.4";
      AN    "M347.5";
      AN    "M348.1";
      AN    "M348.2";
      =     L 15.0;
      A     L 15.0;
      A     "M347.2";
      =     "M348.7";
      A     L 15.0;
      BLD   102;
      =     "M348.6";
NETWORK
TITLE =
      A     "M11.2";
      A     "ToDo";
      A     "M347.3";
      A     "M347.4";
      AN    "M347.5";
      AN    "M348.1";
      AN    "M348.2";
      S     "M346.2";
END_FUNCTION

FUNCTION "FC117 - ERROR TOOL" : VOID	// FC 117
VERSION : 0.1
BEGIN
// (block stored without names or comments; labels and parameter names are numbered)
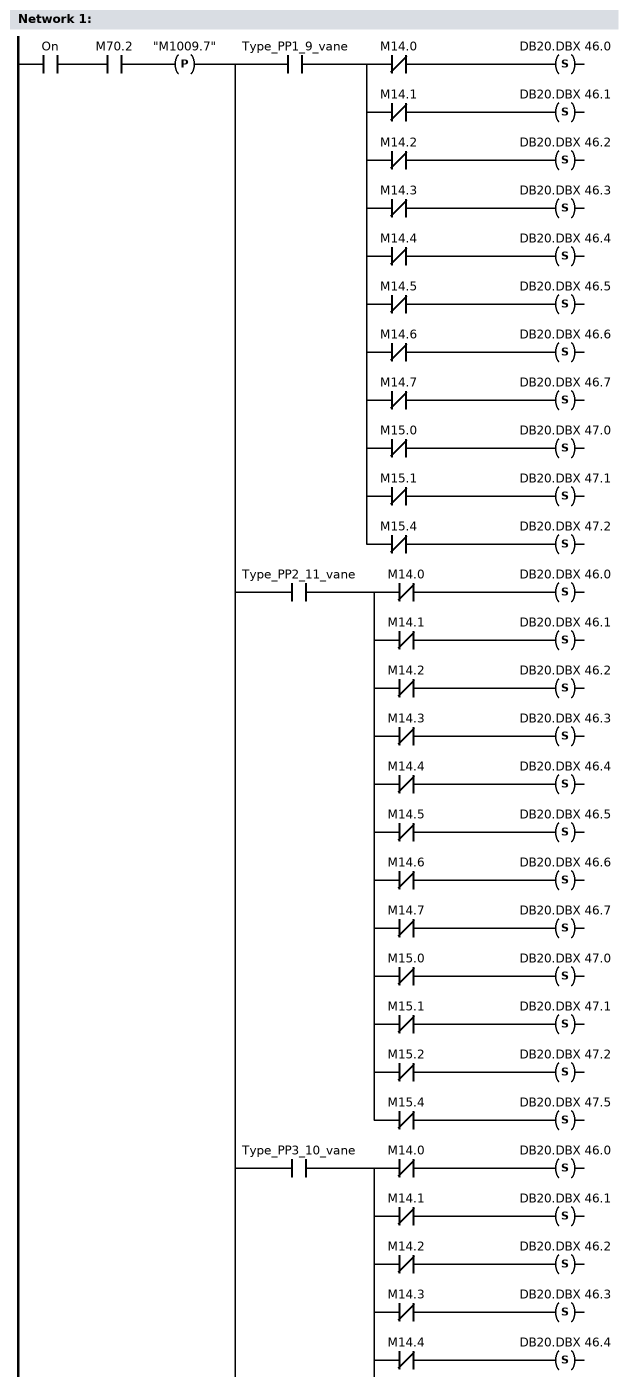
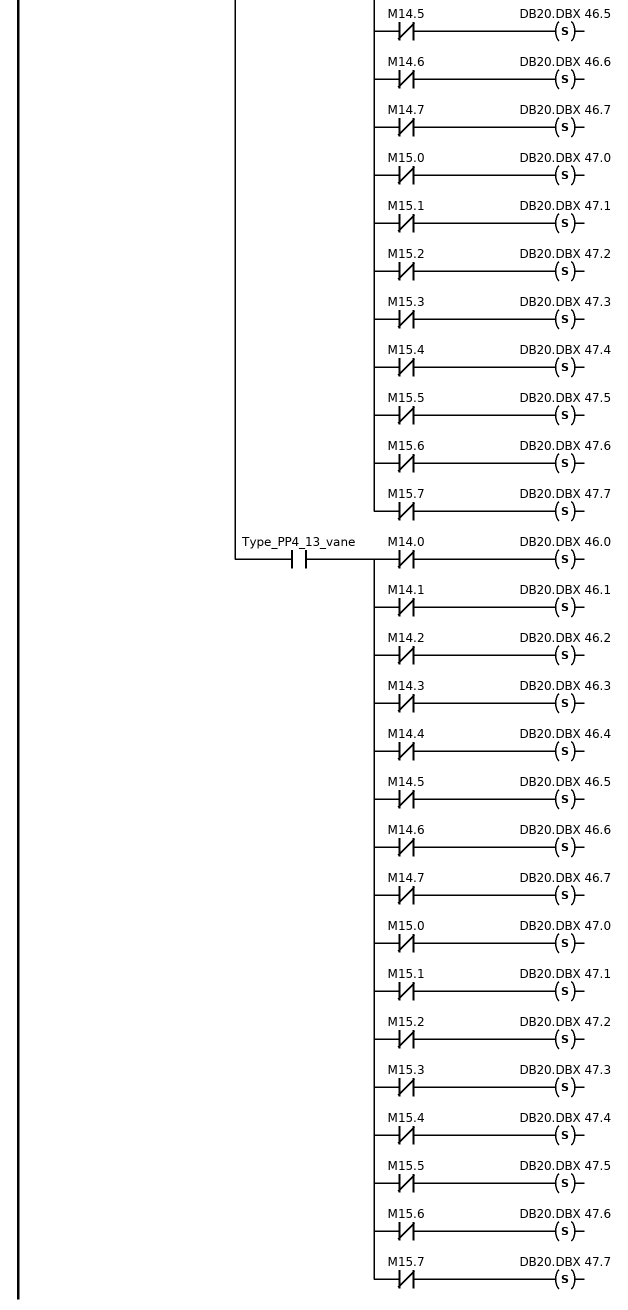
NETWORK
TITLE =
      A     "On";
      A     "M70.2";
      FP    "M1009.7";
      =     L 0.0;
      A     L 0.0;
      A     "Type_PP1_9_vane";
      =     L 0.1;
      A     L 0.1;
      AN    "M14.0";
      S     DB20.DBX 46.0;
      A     L 0.1;
      AN    "M14.1";
      S     DB20.DBX 46.1;
      A     L 0.1;
      AN    "M14.2";
      S     DB20.DBX 46.2;
      A     L 0.1;
      AN    "M14.3";
      S     DB20.DBX 46.3;
      A     L 0.1;
      AN    "M14.4";
      S     DB20.DBX 46.4;
      A     L 0.1;
      AN    "M14.5";
      S     DB20.DBX 46.5;
      A     L 0.1;
      AN    "M14.6";
      S     DB20.DBX 46.6;
      A     L 0.1;
      AN    "M14.7";
      S     DB20.DBX 46.7;
      A     L 0.1;
      AN    "M15.0";
      S     DB20.DBX 47.0;
      A     L 0.1;
      AN    "M15.1";
      S     DB20.DBX 47.1;
      A     L 0.1;
      AN    "M15.4";
      S     DB20.DBX 47.2;
      A     L 0.0;
      A     "Type_PP2_11_vane";
      =     L 0.1;
      A     L 0.1;
      AN    "M14.0";
      S     DB20.DBX 46.0;
      A     L 0.1;
      AN    "M14.1";
      S     DB20.DBX 46.1;
      A     L 0.1;
      AN    "M14.2";
      S     DB20.DBX 46.2;
      A     L 0.1;
      AN    "M14.3";
      S     DB20.DBX 46.3;
      A     L 0.1;
      AN    "M14.4";
      S     DB20.DBX 46.4;
      A     L 0.1;
      AN    "M14.5";
      S     DB20.DBX 46.5;
      A     L 0.1;
      AN    "M14.6";
      S     DB20.DBX 46.6;
      A     L 0.1;
      AN    "M14.7";
      S     DB20.DBX 46.7;
      A     L 0.1;
      AN    "M15.0";
      S     DB20.DBX 47.0;
      A     L 0.1;
      AN    "M15.1";
      S     DB20.DBX 47.1;
      A     L 0.1;
      AN    "M15.2";
      S     DB20.DBX 47.2;
      A     L 0.1;
      AN    "M15.4";
      S     DB20.DBX 47.5;
      A     L 0.0;
      A     "Type_PP3_10_vane";
      =     L 0.1;
      A     L 0.1;
      AN    "M14.0";
      S     DB20.DBX 46.0;
      A     L 0.1;
      AN    "M14.1";
      S     DB20.DBX 46.1;
      A     L 0.1;
      AN    "M14.2";
      S     DB20.DBX 46.2;
      A     L 0.1;
      AN    "M14.3";
      S     DB20.DBX 46.3;
      A     L 0.1;
      AN    "M14.4";
      S     DB20.DBX 46.4;
      A     L 0.1;
      AN    "M14.5";
      S     DB20.DBX 46.5;
      A     L 0.1;
      AN    "M14.6";
      S     DB20.DBX 46.6;
      A     L 0.1;
      AN    "M14.7";
      S     DB20.DBX 46.7;
      A     L 0.1;
      AN    "M15.0";
      S     DB20.DBX 47.0;
      A     L 0.1;
      AN    "M15.1";
      S     DB20.DBX 47.1;
      A     L 0.1;
      AN    "M15.2";
      S     DB20.DBX 47.2;
      A     L 0.1;
      AN    "M15.3";
      S     DB20.DBX 47.3;
      A     L 0.1;
      AN    "M15.4";
      S     DB20.DBX 47.4;
      A     L 0.1;
      AN    "M15.5";
      S     DB20.DBX 47.5;
      A     L 0.1;
      AN    "M15.6";
      S     DB20.DBX 47.6;
      A     L 0.1;
      AN    "M15.7";
      S     DB20.DBX 47.7;
      A     L 0.0;
      A     "Type_PP4_13_vane";
      =     L 0.1;
      A     L 0.1;
      AN    "M14.0";
      S     DB20.DBX 46.0;
      A     L 0.1;
      AN    "M14.1";
      S     DB20.DBX 46.1;
      A     L 0.1;
      AN    "M14.2";
      S     DB20.DBX 46.2;
      A     L 0.1;
      AN    "M14.3";
      S     DB20.DBX 46.3;
      A     L 0.1;
      AN    "M14.4";
      S     DB20.DBX 46.4;
      A     L 0.1;
      AN    "M14.5";
      S     DB20.DBX 46.5;
      A     L 0.1;
      AN    "M14.6";
      S     DB20.DBX 46.6;
      A     L 0.1;
      AN    "M14.7";
      S     DB20.DBX 46.7;
      A     L 0.1;
      AN    "M15.0";
      S     DB20.DBX 47.0;
      A     L 0.1;
      AN    "M15.1";
      S     DB20.DBX 47.1;
      A     L 0.1;
      AN    "M15.2";
      S     DB20.DBX 47.2;
      A     L 0.1;
      AN    "M15.3";
      S     DB20.DBX 47.3;
      A     L 0.1;
      AN    "M15.4";
      S     DB20.DBX 47.4;
      A     L 0.1;
      AN    "M15.5";
      S     DB20.DBX 47.5;
      A     L 0.1;
      AN    "M15.6";
      S     DB20.DBX 47.6;
      A     L 0.1;
      AN    "M15.7";
      S     DB20.DBX 47.7;
END_FUNCTION

FUNCTION "TimeOut" : VOID	// FC 800
AUTHOR : Cellini
FAMILY : GCLib
NAME : TimeOut
VERSION : 1.0
BEGIN
// (block stored without names or comments; labels and parameter names are numbered)
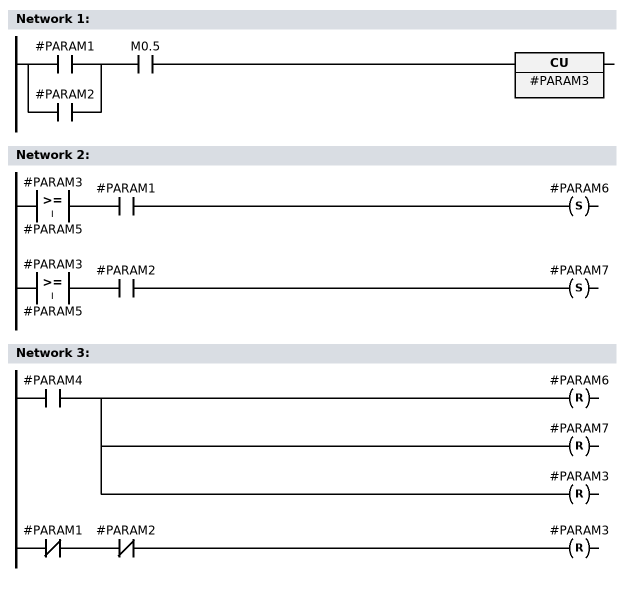
NETWORK
TITLE =
      A     #PARAM1;
      O     #PARAM2;
      A     "M0.5";
      CU    #PARAM3;
NETWORK
TITLE =
      L     #PARAM3;
      L     #PARAM5;
      >=I;
      A     #PARAM1;
      S     #PARAM6;
      L     #PARAM3;
      L     #PARAM5;
      >=I;
      A     #PARAM2;
      S     #PARAM7;
NETWORK
TITLE =
      A     #PARAM4;
      R     #PARAM6;
      R     #PARAM7;
      R     #PARAM3;
      AN    #PARAM1;
      AN    #PARAM2;
      R     #PARAM3;
END_FUNCTION

DATA_BLOCK "DI_Balluff1"	// DB 5
AUTHOR : Salvati
VERSION : 0.0
"BALLUFF"
BEGIN
END_DATA_BLOCK

DATA_BLOCK "DatiOP170B"	// DB 7
AUTHOR : Coletti
FAMILY : GCLib
VERSION : 0.1
BEGIN
// 382 bytes; values not shown
END_DATA_BLOCK

DATA_BLOCK DB 11
VERSION : 0.1
BEGIN
// 38 bytes; values not shown
END_DATA_BLOCK

DATA_BLOCK DB 12
VERSION : 0.1
BEGIN
// 38 bytes; values not shown
END_DATA_BLOCK

DATA_BLOCK DB 13
VERSION : 0.1
BEGIN
// 16 bytes; values not shown
END_DATA_BLOCK

DATA_BLOCK "Timer"	// DB 20
VERSION : 0.1
BEGIN
// 72 bytes; values not shown
END_DATA_BLOCK

DATA_BLOCK "DBWork"	// DB 21
AUTHOR : Coletti
VERSION : 0.1
BEGIN
// 478 bytes; values not shown
END_DATA_BLOCK

DATA_BLOCK "coordinate"	// DB 22
VERSION : 0.1
BEGIN
// 8860 bytes; values not shown
END_DATA_BLOCK

DATA_BLOCK DB 23
VERSION : 0.1
BEGIN
// 2 bytes; values not shown
END_DATA_BLOCK

DATA_BLOCK "DB180"	// DB 180
VERSION : 0.0
"FB24 - Gestione Mov Assi"
BEGIN
END_DATA_BLOCK

DATA_BLOCK "DB181"	// DB 181
VERSION : 0.0
"FB24 - Gestione Mov Assi"
BEGIN
END_DATA_BLOCK

ORGANIZATION_BLOCK "MAIN PROGRAM"	// OB 1
VERSION : 0.1
BEGIN
// (block stored without names or comments; labels and parameter names are numbered)
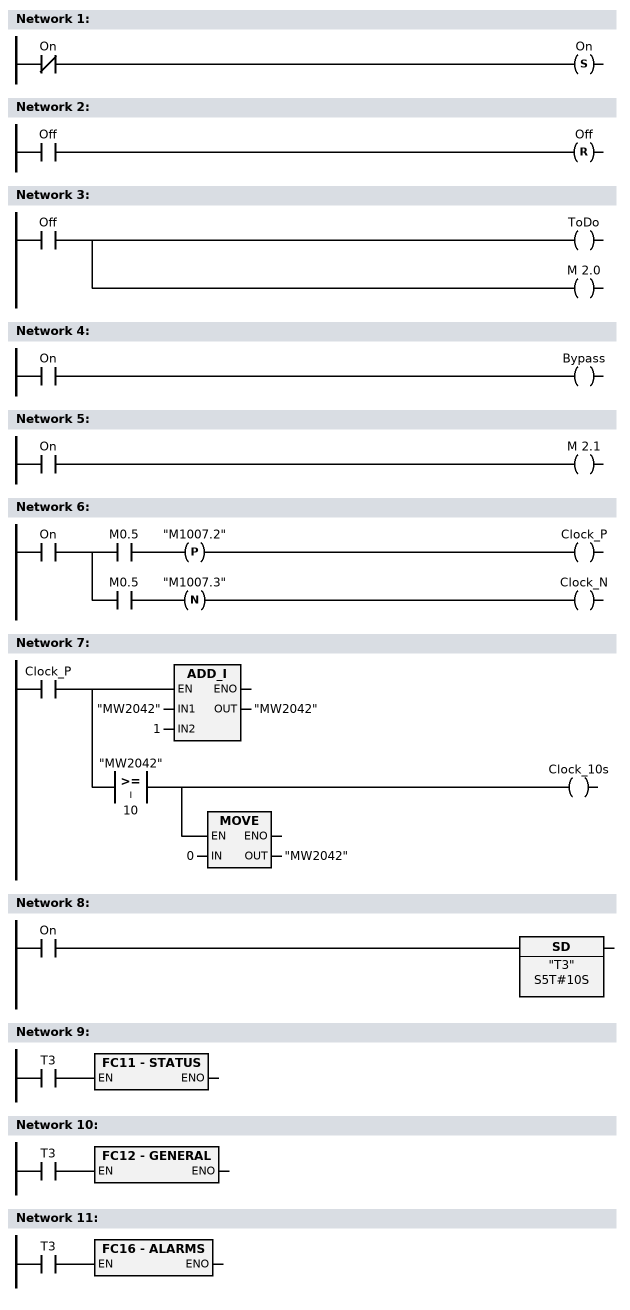
NETWORK
TITLE =
      AN    "On";
      S     "On";
NETWORK
TITLE =
      A     "Off";
      R     "Off";
NETWORK
TITLE =
      A     "Off";
      =     "ToDo";
      =     M 2.0;
NETWORK
TITLE =
      A     "On";
      =     "Bypass";
NETWORK
TITLE =
      A     "On";
      =     M 2.1;
NETWORK
TITLE =
      A     "On";
      =     L 20.0;
      A     L 20.0;
      A     "M0.5";
      FP    "M1007.2";
      =     "Clock_P";
      A     L 20.0;
      A     "M0.5";
      FN    "M1007.3";
      =     "Clock_N";
NETWORK
TITLE =
      A     "Clock_P";
      =     L 20.0;
      A     L 20.0;
      JNB   M001;
      L     "MW2042";
      L     1;
      +I;
      T     "MW2042";
M001: NOP   0;
      A     L 20.0;
      A(;
      L     "MW2042";
      L     10;
      >=I;
      );
      =     L 20.1;
      A     L 20.1;
      BLD   102;
      =     "Clock_10s";
      A     L 20.1;
      JNB   M002;
      L     0;
      T     "MW2042";
M002: NOP   0;
NETWORK
TITLE =
      A     "On";
      L     S5T#10S;
      SD    "T3";
NETWORK
TITLE =
      A     "T3";
      JNB   M003;
      CALL  "FC11 - STATUS";
M003: NOP   0;
NETWORK
TITLE =
      A     "T3";
      JNB   M004;
      CALL  "FC12 - GENERAL";
M004: NOP   0;
NETWORK
TITLE =
      A     "T3";
      JNB   M005;
      CALL  "FC16 - ALARMS";
M005: NOP   0;
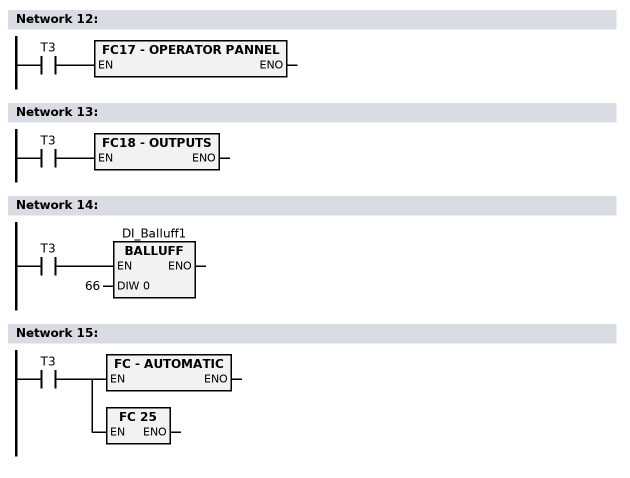
NETWORK
TITLE =
      A     "T3";
      JNB   M006;
      CALL  "FC17 - OPERATOR PANNEL";
M006: NOP   0;
NETWORK
TITLE =
      A     "T3";
      JNB   M007;
      CALL  "FC18 - OUTPUTS";
M007: NOP   0;
NETWORK
TITLE =
      A     "T3";
      JNB   M008;
      CALL  "BALLUFF" , "DI_Balluff1" (
           DIW 0                    := 66);
M008: NOP   0;
NETWORK
TITLE =
      A     "T3";
      =     L 20.0;
      A     L 20.0;
      JNB   M009;
      CALL  "FC - AUTOMATIC";
M009: NOP   0;
      A     L 20.0;
      JNB   M010;
      CALL  FC 25;
M010: NOP   0;
END_ORGANIZATION_BLOCK

ORGANIZATION_BLOCK "I/O_FLT1"	// OB 82
VERSION : 1.0
BEGIN
// (block stored without names or comments; labels and parameter names are numbered)
NETWORK
TITLE =
END_ORGANIZATION_BLOCK

ORGANIZATION_BLOCK "RACK_FLT"	// OB 86
VERSION : 0.1
BEGIN
// (block stored without names or comments; labels and parameter names are numbered)
NETWORK
TITLE =
END_ORGANIZATION_BLOCK

ORGANIZATION_BLOCK "COMPLETE RESTART"	// OB 100
VERSION : 0.1
BEGIN
// (block stored without names or comments; labels and parameter names are numbered)
